gfCNCPoint4[24000] = {X 138.7499, Y 45.9791, Z -6.3333, A 0.000, B 0.000, C 0.000 }
gfCNCPoint4[24001] = {X 138.6396, Y 45.0000, Z -6.3333, A 0.000, B 0.000, C 0.000 }
gfCNCPoint4[24002] = {X 138.6400, Y 44.1483, Z -6.3333, A 0.000, B 0.000, C 0.000 }
gfCNCPoint4[24003] = {X 138.7505, Y 43.2275, Z -6.3333, A 0.000, B 0.000, C 0.000 }
gfCNCPoint4[24004] = {X 139.0514, Y 42.3503, Z -6.3333, A 0.000, B 0.000, C 0.000 }
gfCNCPoint4[24005] = {X 139.5295, Y 41.5556, Z -6.3333, A 0.000, B 0.000, C 0.000 }
gfCNCPoint4[24006] = {X 140.1636, Y 40.8789, Z -6.3333, A 0.000, B 0.000, C 0.000 }
gfCNCPoint4[24007] = {X 140.1636, Y 19.9580, Z -6.3333, A 0.000, B 0.000, C 0.000 }
gfCNCPoint4[24008] = {X 137.4658, Y 19.9576, Z -6.3333, A 0.000, B 0.000, C 0.000 }
gfCNCPoint4[24009] = {X 136.9182, Y 20.6078, Z -6.3333, A 0.000, B 0.000, C 0.000 }
gfCNCPoint4[24010] = {X 136.2556, Y 21.1406, Z -6.3333, A 0.000, B 0.000, C 0.000 }
gfCNCPoint4[24011] = {X 135.5030, Y 21.5361, Z -6.3333, A 0.000, B 0.000, C 0.000 }
gfCNCPoint4[24012] = {X 134.6884, Y 21.7794, Z -6.3333, A 0.000, B 0.000, C 0.000 }
gfCNCPoint4[24013] = {X 133.8422, Y 21.8615, Z -6.3333, A 0.000, B 0.000, C 0.000 }
gfCNCPoint4[24014] = {X 133.2006, Y 21.8615, Z -6.3333, A 0.000, B 0.000, C 0.000 }
gfCNCPoint4[24015] = {X 132.2215, Y 21.7512, Z -6.3333, A 0.000, B 0.000, C 0.000 }
gfCNCPoint4[24016] = {X 131.2916, Y 21.4258, Z -6.3333, A 0.000, B 0.000, C 0.000 }
gfCNCPoint4[24017] = {X 130.4573, Y 20.9016, Z -6.3333, A 0.000, B 0.000, C 0.000 }
gfCNCPoint4[24018] = {X 129.7606, Y 20.2049, Z -6.3333, A 0.000, B 0.000, C 0.000 }
gfCNCPoint4[24019] = {X 129.2364, Y 19.3706, Z -6.3333, A 0.000, B 0.000, C 0.000 }
gfCNCPoint4[24020] = {X 128.9110, Y 18.4406, Z -6.3333, A 0.000, B 0.000, C 0.000 }
gfCNCPoint4[24021] = {X 128.8006, Y 17.4615, Z -6.3333, A 0.000, B 0.000, C 0.000 }
gfCNCPoint4[24022] = {X 128.8006, Y 10.4835, Z -6.3333, A 0.000, B 0.000, C 0.000 }
gfCNCPoint4[24023] = {X 128.8808, Y 9.6474, Z -6.3333, A 0.000, B 0.000, C 0.000 }
gfCNCPoint4[24024] = {X 129.1184, Y 8.8418, Z -6.3333, A 0.000, B 0.000, C 0.000 }
gfCNCPoint4[24025] = {X 129.5047, Y 8.0960, Z -6.3333, A 0.000, B 0.000, C 0.000 }
gfCNCPoint4[24026] = {X 130.0257, Y 7.4372, Z -6.3333, A 0.000, B 0.000, C 0.000 }
gfCNCPoint4[24027] = {X 129.6794, Y 7.1049, Z -6.3333, A 0.000, B 0.000, C 0.000 }
gfCNCPoint4[24028] = {X 102.4337, Y 7.1049, Z -6.3333, A 0.000, B 0.000, C 0.000 }
gfCNCPoint4[24029] = {X 102.4337, Y 11.9049, Z -6.3333, A 0.000, B 0.000, C 0.000 }
gfCNCPoint4[24030] = {X 101.3242, Y 11.9049, Z -6.3333, A 0.000, B 0.000, C 0.000 }
gfCNCPoint4[24031] = {X 101.3283, Y 12.0458, Z -6.3333, A 0.000, B 0.000, C 0.000 }
gfCNCPoint4[24032] = {X 101.3297, Y 12.1868, Z -6.3333, A 0.000, B 0.000, C 0.000 }
gfCNCPoint4[24033] = {X 101.3293, Y 13.0462, Z -6.3333, A 0.000, B 0.000, C 0.000 }
gfCNCPoint4[24034] = {X 101.2275, Y 14.1932, Z -6.3333, A 0.000, B 0.000, C 0.000 }
gfCNCPoint4[24035] = {X 100.9461, Y 15.3098, Z -6.3333, A 0.000, B 0.000, C 0.000 }
gfCNCPoint4[24036] = {X 101.0403, Y 15.5443, Z -6.3333, A 0.000, B 0.000, C 0.000 }
gfCNCPoint4[24037] = {X 101.8677, Y 17.5951, Z -6.3333, A 0.000, B 0.000, C 0.000 }
gfCNCPoint4[24038] = {X 102.7996, Y 15.2734, Z -6.3333, A 0.000, B 0.000, C 0.000 }
gfCNCPoint4[24039] = {X 102.5263, Y 14.1685, Z -6.3333, A 0.000, B 0.000, C 0.000 }
gfCNCPoint4[24040] = {X 102.4285, Y 13.0344, Z -6.3333, A 0.000, B 0.000, C 0.000 }
gfCNCPoint4[24041] = {X 102.4283, Y 12.1868, Z -6.3333, A 0.000, B 0.000, C 0.000 }
gfCNCPoint4[24042] = {X 102.4296, Y 12.0458, Z -6.3333, A 0.000, B 0.000, C 0.000 }
gfCNCPoint4[24043] = {X 102.4337, Y 11.9049, Z -6.3333, A 0.000, B 0.000, C 0.000 }
gfCNCPoint4[24044] = {X 102.4337, Y 9.5049, Z -6.3333, A 0.000, B 0.000, C 0.000 }
gfCNCPoint4[24045] = {X 98.1266, Y 9.5049, Z -6.3333, A 0.000, B 0.000, C 0.000 }
gfCNCPoint4[24046] = {X 98.5429, Y 10.2828, Z -6.3333, A 0.000, B 0.000, C 0.000 }
gfCNCPoint4[24047] = {X 98.8123, Y 11.1229, Z -6.3333, A 0.000, B 0.000, C 0.000 }
gfCNCPoint4[24048] = {X 98.9260, Y 11.9978, Z -6.3333, A 0.000, B 0.000, C 0.000 }
gfCNCPoint4[24049] = {X 98.9288, Y 12.0923, Z -6.3333, A 0.000, B 0.000, C 0.000 }
gfCNCPoint4[24050] = {X 98.9297, Y 12.1868, Z -6.3333, A 0.000, B 0.000, C 0.000 }
gfCNCPoint4[24051] = {X 98.9294, Y 13.0237, Z -6.3333, A 0.000, B 0.000, C 0.000 }
gfCNCPoint4[24052] = {X 98.8590, Y 13.8055, Z -6.3333, A 0.000, B 0.000, C 0.000 }
gfCNCPoint4[24053] = {X 98.6641, Y 14.5659, Z -6.3333, A 0.000, B 0.000, C 0.000 }
gfCNCPoint4[24054] = {X 98.3499, Y 15.2851, Z -6.3333, A 0.000, B 0.000, C 0.000 }
gfCNCPoint4[24055] = {X 98.8140, Y 16.4405, Z -6.3333, A 0.000, B 0.000, C 0.000 }
gfCNCPoint4[24056] = {X 101.8734, Y 24.0244, Z -6.3333, A 0.000, B 0.000, C 0.000 }
gfCNCPoint4[24057] = {X 103.9028, Y 18.9676, Z -6.3333, A 0.000, B 0.000, C 0.000 }
gfCNCPoint4[24058] = {X 105.3927, Y 15.2562, Z -6.3333, A 0.000, B 0.000, C 0.000 }
gfCNCPoint4[24059] = {X 105.0867, Y 14.5450, Z -6.3333, A 0.000, B 0.000, C 0.000 }
gfCNCPoint4[24060] = {X 104.8970, Y 13.7943, Z -6.3333, A 0.000, B 0.000, C 0.000 }
gfCNCPoint4[24061] = {X 104.8285, Y 13.0231, Z -6.3333, A 0.000, B 0.000, C 0.000 }
gfCNCPoint4[24062] = {X 104.8283, Y 12.1868, Z -6.3333, A 0.000, B 0.000, C 0.000 }
gfCNCPoint4[24063] = {X 104.8292, Y 12.0923, Z -6.3333, A 0.000, B 0.000, C 0.000 }
gfCNCPoint4[24064] = {X 104.8319, Y 11.9978, Z -6.3333, A 0.000, B 0.000, C 0.000 }
gfCNCPoint4[24065] = {X 104.9457, Y 11.1229, Z -6.3333, A 0.000, B 0.000, C 0.000 }
gfCNCPoint4[24066] = {X 105.2150, Y 10.2828, Z -6.3333, A 0.000, B 0.000, C 0.000 }
gfCNCPoint4[24067] = {X 105.6313, Y 9.5049, Z -6.3333, A 0.000, B 0.000, C 0.000 }
gfCNCPoint4[24068] = {X 102.4337, Y 9.5049, Z -6.3333, A 0.000, B 0.000, C 0.000 }
gfCNCPoint4[24069] = {X 102.4337, Y 7.1049, Z -6.3333, A 0.000, B 0.000, C 0.000 }
gfCNCPoint4[24070] = {X 64.8349, Y 7.1049, Z -6.3333, A 0.000, B 0.000, C 0.000 }
gfCNCPoint4[24071] = {X 65.5946, Y 8.0241, Z -6.3333, A 0.000, B 0.000, C 0.000 }
gfCNCPoint4[24072] = {X 66.1940, Y 9.0549, Z -6.3333, A 0.000, B 0.000, C 0.000 }
gfCNCPoint4[24073] = {X 66.6171, Y 10.1698, Z -6.3333, A 0.000, B 0.000, C 0.000 }
gfCNCPoint4[24074] = {X 66.8305, Y 11.1683, Z -6.3333, A 0.000, B 0.000, C 0.000 }
gfCNCPoint4[24075] = {X 66.9021, Y 12.1868, Z -6.3333, A 0.000, B 0.000, C 0.000 }
gfCNCPoint4[24076] = {X 66.9018, Y 13.0462, Z -6.3333, A 0.000, B 0.000, C 0.000 }
gfCNCPoint4[24077] = {X 66.7773, Y 14.3204, Z -6.3333, A 0.000, B 0.000, C 0.000 }
gfCNCPoint4[24078] = {X 66.4315, Y 15.5530, Z -6.3333, A 0.000, B 0.000, C 0.000 }
gfCNCPoint4[24079] = {X 74.9126, Y 38.2401, Z -6.3333, A 0.000, B 0.000, C 0.000 }
gfCNCPoint4[24080] = {X 75.8046, Y 38.9749, Z -6.3333, A 0.000, B 0.000, C 0.000 }
gfCNCPoint4[24081] = {X 76.5691, Y 39.8416, Z -6.3333, A 0.000, B 0.000, C 0.000 }
gfCNCPoint4[24082] = {X 77.1868, Y 40.8184, Z -6.3333, A 0.000, B 0.000, C 0.000 }
gfCNCPoint4[24083] = {X 77.6421, Y 41.8806, Z -6.3333, A 0.000, B 0.000, C 0.000 }
gfCNCPoint4[24084] = {X 77.9236, Y 43.0014, Z -6.3333, A 0.000, B 0.000, C 0.000 }
gfCNCPoint4[24085] = {X 78.0243, Y 44.1527, Z -6.3333, A 0.000, B 0.000, C 0.000 }
gfCNCPoint4[24086] = {X 78.0245, Y 45.0000, Z -6.3333, A 0.000, B 0.000, C 0.000 }
gfCNCPoint4[24087] = {X 77.9139, Y 46.2642, Z -6.3333, A 0.000, B 0.000, C 0.000 }
gfCNCPoint4[24088] = {X 77.5854, Y 47.4899, Z -6.3333, A 0.000, B 0.000, C 0.000 }
gfCNCPoint4[24089] = {X 77.0491, Y 48.6400, Z -6.3333, A 0.000, B 0.000, C 0.000 }
gfCNCPoint4[24090] = {X 76.3213, Y 49.6795, Z -6.3333, A 0.000, B 0.000, C 0.000 }
gfCNCPoint4[24091] = {X 75.4240, Y 50.5768, Z -6.3333, A 0.000, B 0.000, C 0.000 }
gfCNCPoint4[24092] = {X 74.3845, Y 51.3047, Z -6.3333, A 0.000, B 0.000, C 0.000 }
gfCNCPoint4[24093] = {X 73.2344, Y 51.8410, Z -6.3333, A 0.000, B 0.000, C 0.000 }
gfCNCPoint4[24094] = {X 72.0086, Y 52.1694, Z -6.3333, A 0.000, B 0.000, C 0.000 }
gfCNCPoint4[24095] = {X 70.7445, Y 52.2800, Z -6.3333, A 0.000, B 0.000, C 0.000 }
gfCNCPoint4[24096] = {X 64.1851, Y 52.2800, Z -6.3333, A 0.000, B 0.000, C 0.000 }
gfCNCPoint4[24097] = {X 62.9397, Y 52.1727, Z -6.3333, A 0.000, B 0.000, C 0.000 }
gfCNCPoint4[24098] = {X 61.7311, Y 51.8539, Z -6.3333, A 0.000, B 0.000, C 0.000 }
gfCNCPoint4[24099] = {X 60.5947, Y 51.3330, Z -6.3333, A 0.000, B 0.000, C 0.000 }
gfCNCPoint4[24100] = {X 59.5643, Y 50.6255, Z -6.3333, A 0.000, B 0.000, C 0.000 }
gfCNCPoint4[24101] = {X 58.6700, Y 49.7521, Z -6.3333, A 0.000, B 0.000, C 0.000 }
gfCNCPoint4[24102] = {X 57.9384, Y 48.7385, Z -6.3333, A 0.000, B 0.000, C 0.000 }
gfCNCPoint4[24103] = {X 57.3706, Y 47.5614, Z -6.3333, A 0.000, B 0.000, C 0.000 }
gfCNCPoint4[24104] = {X 57.0225, Y 46.3017, Z -6.3333, A 0.000, B 0.000, C 0.000 }
gfCNCPoint4[24105] = {X 56.9051, Y 45.0000, Z -6.3333, A 0.000, B 0.000, C 0.000 }
gfCNCPoint4[24106] = {X 56.9052, Y 44.1969, Z -6.3333, A 0.000, B 0.000, C 0.000 }
gfCNCPoint4[24107] = {X 56.9289, Y 43.6212, Z -6.3333, A 0.000, B 0.000, C 0.000 }
gfCNCPoint4[24108] = {X 56.9981, Y 43.0492, Z -6.3333, A 0.000, B 0.000, C 0.000 }
gfCNCPoint4[24109] = {X 54.7600, Y 43.0492, Z -6.3333, A 0.000, B 0.000, C 0.000 }
gfCNCPoint4[24110] = {X 54.8275, Y 43.6012, Z -6.3333, A 0.000, B 0.000, C 0.000 }
gfCNCPoint4[24111] = {X 54.8528, Y 44.1567, Z -6.3333, A 0.000, B 0.000, C 0.000 }
gfCNCPoint4[24112] = {X 54.8529, Y 45.0000, Z -6.3333, A 0.000, B 0.000, C 0.000 }
gfCNCPoint4[24113] = {X 54.7356, Y 46.3017, Z -6.3333, A 0.000, B 0.000, C 0.000 }
gfCNCPoint4[24114] = {X 54.3875, Y 47.5614, Z -6.3333, A 0.000, B 0.000, C 0.000 }
gfCNCPoint4[24115] = {X 53.8197, Y 48.7385, Z -6.3333, A 0.000, B 0.000, C 0.000 }
gfCNCPoint4[24116] = {X 53.0880, Y 49.7521, Z -6.3333, A 0.000, B 0.000, C 0.000 }
gfCNCPoint4[24117] = {X 52.1938, Y 50.6255, Z -6.3333, A 0.000, B 0.000, C 0.000 }
gfCNCPoint4[24118] = {X 51.1633, Y 51.3330, Z -6.3333, A 0.000, B 0.000, C 0.000 }
gfCNCPoint4[24119] = {X 50.0270, Y 51.8539, Z -6.3333, A 0.000, B 0.000, C 0.000 }
gfCNCPoint4[24120] = {X 48.8183, Y 52.1727, Z -6.3333, A 0.000, B 0.000, C 0.000 }
gfCNCPoint4[24121] = {X 47.5729, Y 52.2800, Z -6.3333, A 0.000, B 0.000, C 0.000 }
gfCNCPoint4[24122] = {X 40.6393, Y 52.2800, Z -6.3333, A 0.000, B 0.000, C 0.000 }
gfCNCPoint4[24123] = {X 39.4476, Y 52.1818, Z -6.3333, A 0.000, B 0.000, C 0.000 }
gfCNCPoint4[24124] = {X 38.2881, Y 51.8899, Z -6.3333, A 0.000, B 0.000, C 0.000 }
gfCNCPoint4[24125] = {X 37.1919, Y 51.4120, Z -6.3333, A 0.000, B 0.000, C 0.000 }
gfCNCPoint4[24126] = {X 36.1888, Y 50.7612, Z -6.3333, A 0.000, B 0.000, C 0.000 }
gfCNCPoint4[24127] = {X 35.3058, Y 49.9550, Z -6.3333, A 0.000, B 0.000, C 0.000 }
gfCNCPoint4[24128] = {X 34.8234, Y 50.4196, Z -6.3333, A 0.000, B 0.000, C 0.000 }
gfCNCPoint4[24129] = {X 34.3150, Y 50.8555, Z -6.3333, A 0.000, B 0.000, C 0.000 }
gfCNCPoint4[24130] = {X 33.7788, Y 51.2890, Z -6.3333, A 0.000, B 0.000, C 0.000 }
gfCNCPoint4[24131] = {X 32.5198, Y 52.1756, Z -6.3333, A 0.000, B 0.000, C 0.000 }
gfCNCPoint4[24132] = {X 31.1545, Y 52.8879, Z -6.3333, A 0.000, B 0.000, C 0.000 }
gfCNCPoint4[24133] = {X 29.7070, Y 53.4132, Z -6.3333, A 0.000, B 0.000, C 0.000 }
gfCNCPoint4[24134] = {X 28.2028, Y 53.7423, Z -6.3333, A 0.000, B 0.000, C 0.000 }
gfCNCPoint4[24135] = {X 26.6682, Y 53.8696, Z -6.3333, A 0.000, B 0.000, C 0.000 }
gfCNCPoint4[24136] = {X 24.3194, Y 54.9126, Z -6.3333, A 0.000, B 0.000, C 0.000 }
gfCNCPoint4[24137] = {X 21.9033, Y 55.7884, Z -6.3333, A 0.000, B 0.000, C 0.000 }
gfCNCPoint4[24138] = {X 19.5297, Y 56.4643, Z -6.3333, A 0.000, B 0.000, C 0.000 }
gfCNCPoint4[24139] = {X 17.1086, Y 56.9430, Z -6.3333, A 0.000, B 0.000, C 0.000 }
gfCNCPoint4[24140] = {X 14.6564, Y 57.2213, Z -6.3333, A 0.000, B 0.000, C 0.000 }
gfCNCPoint4[24141] = {X 12.1897, Y 57.2974, Z -6.3333, A 0.000, B 0.000, C 0.000 }
gfCNCPoint4[24142] = {X 9.7250, Y 57.1707, Z -6.3333, A 0.000, B 0.000, C 0.000 }
gfCNCPoint4[24143] = {X 8.4102, Y 57.0194, Z -6.3333, A 0.000, B 0.000, C 0.000 }
gfCNCPoint4[24144] = {X 7.1034, Y 56.8104, Z -6.3333, A 0.000, B 0.000, C 0.000 }
gfCNCPoint4[24145] = {X 7.1034, Y 92.8951, Z -6.3333, A 0.000, B 0.000, C 0.000 }
gfCNCPoint4[24146] = {X 116.2646, Y 92.8951, Z -6.3333, A 0.000, B 0.000, C 0.000 }
gfCNCPoint4[24147] = {X 116.9710, Y 91.6587, Z -6.3333, A 0.000, B 0.000, C 0.000 }
gfCNCPoint4[24148] = {X 117.8511, Y 90.5393, Z -6.3333, A 0.000, B 0.000, C 0.000 }
gfCNCPoint4[24149] = {X 118.8860, Y 89.5612, Z -6.3333, A 0.000, B 0.000, C 0.000 }
gfCNCPoint4[24150] = {X 120.0531, Y 88.7455, Z -6.3333, A 0.000, B 0.000, C 0.000 }
gfCNCPoint4[24151] = {X 121.3272, Y 88.1097, Z -6.3333, A 0.000, B 0.000, C 0.000 }
gfCNCPoint4[24152] = {X 122.6809, Y 87.6678, Z -6.3333, A 0.000, B 0.000, C 0.000 }
gfCNCPoint4[24153] = {X 124.0847, Y 87.4293, Z -6.3333, A 0.000, B 0.000, C 0.000 }
gfCNCPoint4[24154] = {X 124.5363, Y 87.3610, Z -6.3333, A 0.000, B 0.000, C 0.000 }
gfCNCPoint4[24155] = {X 125.0288, Y 86.8573, Z -6.3333, A 0.000, B 0.000, C 0.000 }
gfCNCPoint4[24156] = {X 125.5072, Y 86.3401, Z -6.3333, A 0.000, B 0.000, C 0.000 }
gfCNCPoint4[24157] = {X 149.6585, Y 59.8188, Z -6.3333, A 0.000, B 0.000, C 0.000 }
gfCNCPoint4[24158] = {X 149.6295, Y 59.4063, Z -6.3333, A 0.000, B 0.000, C 0.000 }
gfCNCPoint4[24159] = {X 149.6181, Y 58.9930, Z -6.3333, A 0.000, B 0.000, C 0.000 }
gfCNCPoint4[24160] = {X 149.6180, Y 58.0000, Z -6.3333, A 0.000, B 0.000, C 0.000 }
gfCNCPoint4[24161] = {X 149.6915, Y 56.8093, Z -6.3333, A 0.000, B 0.000, C 0.000 }
gfCNCPoint4[24162] = {X 149.9109, Y 55.6367, Z -6.3333, A 0.000, B 0.000, C 0.000 }
gfCNCPoint4[24163] = {X 150.2729, Y 54.5000, Z -6.3333, A 0.000, B 0.000, C 0.000 }
gfCNCPoint4[24164] = {X 150.7719, Y 53.4164, Z -6.3333, A 0.000, B 0.000, C 0.000 }
gfCNCPoint4[24165] = {X 151.5117, Y 52.2488, Z -6.3333, A 0.000, B 0.000, C 0.000 }
gfCNCPoint4[24166] = {X 152.4103, Y 51.1984, Z -6.3333, A 0.000, B 0.000, C 0.000 }
gfCNCPoint4[24167] = {X 153.4493, Y 50.2867, Z -6.3333, A 0.000, B 0.000, C 0.000 }
gfCNCPoint4[24168] = {X 154.6075, Y 49.5323, Z -6.3333, A 0.000, B 0.000, C 0.000 }
gfCNCPoint4[24169] = {X 155.8614, Y 48.9505, Z -6.3333, A 0.000, B 0.000, C 0.000 }
gfCNCPoint4[24170] = {X 157.1854, Y 48.5533, Z -6.3333, A 0.000, B 0.000, C 0.000 }
gfCNCPoint4[24171] = {X 158.2353, Y 48.3785, Z -6.3333, A 0.000, B 0.000, C 0.000 }
gfCNCPoint4[24172] = {X 159.2980, Y 48.3200, Z -6.3333, A 0.000, B 0.000, C 0.000 }
gfCNCPoint4[24173] = {X 176.3020, Y 48.3200, Z -6.3333, A 0.000, B 0.000, C 0.000 }
gfCNCPoint4[24174] = {X 174.9301, Y 47.4865, Z -6.3333, A 0.000, B 0.000, C 0.000 }
gfCNCPoint4[24175] = {X 173.6422, Y 46.5284, Z -6.3333, A 0.000, B 0.000, C 0.000 }
gfCNCPoint4[24176] = {X 172.5424, Y 45.5341, Z -6.3333, A 0.000, B 0.000, C 0.000 }
gfCNCPoint4[24177] = {X 171.5575, Y 44.4259, Z -6.3333, A 0.000, B 0.000, C 0.000 }
gfCNCPoint4[24178] = {X 170.5960, Y 43.0508, Z -6.3333, A 0.000, B 0.000, C 0.000 }
gfCNCPoint4[24179] = {X 169.8114, Y 41.5676, Z -6.3333, A 0.000, B 0.000, C 0.000 }
gfCNCPoint4[24180] = {X 169.2155, Y 39.9990, Z -6.3333, A 0.000, B 0.000, C 0.000 }
gfCNCPoint4[24181] = {X 168.8176, Y 38.3690, Z -6.3333, A 0.000, B 0.000, C 0.000 }
gfCNCPoint4[24182] = {X 168.7074, Y 37.6766, Z -6.3333, A 0.000, B 0.000, C 0.000 }
gfCNCPoint4[24183] = {X 168.5427, Y 36.0108, Z -6.3333, A 0.000, B 0.000, C 0.000 }
gfCNCPoint4[24184] = {X 168.5600, Y 34.3369, Z -6.3333, A 0.000, B 0.000, C 0.000 }
gfCNCPoint4[24185] = {X 168.7592, Y 32.6747, Z -6.3333, A 0.000, B 0.000, C 0.000 }
gfCNCPoint4[24186] = {X 169.1378, Y 31.0441, Z -6.3333, A 0.000, B 0.000, C 0.000 }
gfCNCPoint4[24187] = {X 169.6914, Y 29.4643, Z -6.3333, A 0.000, B 0.000, C 0.000 }
gfCNCPoint4[24188] = {X 170.2633, Y 28.2675, Z -6.3333, A 0.000, B 0.000, C 0.000 }
gfCNCPoint4[24189] = {X 170.9701, Y 27.1451, Z -6.3333, A 0.000, B 0.000, C 0.000 }
gfCNCPoint4[24190] = {X 171.8024, Y 26.1122, Z -6.3333, A 0.000, B 0.000, C 0.000 }
gfCNCPoint4[24191] = {X 172.7488, Y 25.1829, Z -6.3333, A 0.000, B 0.000, C 0.000 }
gfCNCPoint4[24192] = {X 173.7967, Y 24.3696, Z -6.3333, A 0.000, B 0.000, C 0.000 }
gfCNCPoint4[24193] = {X 173.0267, Y 23.7514, Z -6.3333, A 0.000, B 0.000, C 0.000 }
gfCNCPoint4[24194] = {X 172.3970, Y 22.9909, Z -6.3333, A 0.000, B 0.000, C 0.000 }
gfCNCPoint4[24195] = {X 171.9332, Y 22.1192, Z -6.3333, A 0.000, B 0.000, C 0.000 }
gfCNCPoint4[24196] = {X 169.3220, Y 15.7237, Z -6.3333, A 0.000, B 0.000, C 0.000 }
gfCNCPoint4[24197] = {X 169.1088, Y 15.0753, Z -6.3333, A 0.000, B 0.000, C 0.000 }
gfCNCPoint4[24198] = {X 168.9882, Y 14.4035, Z -6.3333, A 0.000, B 0.000, C 0.000 }
gfCNCPoint4[24199] = {X 168.9599, Y 13.8791, Z -6.3333, A 0.000, B 0.000, C 0.000 }
gfCNCPoint4[24200] = {X 168.9882, Y 13.3548, Z -6.3333, A 0.000, B 0.000, C 0.000 }
gfCNCPoint4[24201] = {X 169.1590, Y 12.4995, Z -6.3333, A 0.000, B 0.000, C 0.000 }
gfCNCPoint4[24202] = {X 169.4794, Y 11.6882, Z -6.3333, A 0.000, B 0.000, C 0.000 }
gfCNCPoint4[24203] = {X 169.9391, Y 10.9470, Z -6.3333, A 0.000, B 0.000, C 0.000 }
gfCNCPoint4[24204] = {X 170.6136, Y 10.2179, Z -6.3333, A 0.000, B 0.000, C 0.000 }
gfCNCPoint4[24205] = {X 171.4217, Y 9.6404, Z -6.3333, A 0.000, B 0.000, C 0.000 }
gfCNCPoint4[24206] = {X 172.0576, Y 9.2779, Z -6.3333, A 0.000, B 0.000, C 0.000 }
gfCNCPoint4[24207] = {X 172.9925, Y 8.8772, Z -6.3333, A 0.000, B 0.000, C 0.000 }
gfCNCPoint4[24208] = {X 173.9903, Y 8.6790, Z -6.3333, A 0.000, B 0.000, C 0.000 }
gfCNCPoint4[24209] = {X 175.0074, Y 8.6919, Z -6.3333, A 0.000, B 0.000, C 0.000 }
gfCNCPoint4[24210] = {X 175.9998, Y 8.9154, Z -6.3333, A 0.000, B 0.000, C 0.000 }
gfCNCPoint4[24211] = {X 176.9280, Y 8.5206, Z -6.3333, A 0.000, B 0.000, C 0.000 }
gfCNCPoint4[24212] = {X 179.1598, Y 7.6998, Z -6.3333, A 0.000, B 0.000, C 0.000 }
gfCNCPoint4[24213] = {X 181.4622, Y 7.1049, Z -6.3333, A 0.000, B 0.000, C 0.000 }
gfCNCPoint4[24214] = {X 168.0206, Y 7.1049, Z -6.3333, A 0.000, B 0.000, C 0.000 }
gfCNCPoint4[24215] = {X 168.0206, Y 4.7049, Z -6.3333, A 0.000, B 0.000, C 0.000 }
gfCNCPoint4[24216] = {X 155.1591, Y 4.7049, Z -6.3333, A 0.000, B 0.000, C 0.000 }
gfCNCPoint4[24217] = {X 155.1591, Y 7.1049, Z -6.3333, A 0.000, B 0.000, C 0.000 }
gfCNCPoint4[24218] = {X 137.3636, Y 7.1049, Z -6.3333, A 0.000, B 0.000, C 0.000 }
gfCNCPoint4[24219] = {X 137.5332, Y 7.2910, Z -6.3333, A 0.000, B 0.000, C 0.000 }
gfCNCPoint4[24220] = {X 137.6930, Y 7.4857, Z -6.3333, A 0.000, B 0.000, C 0.000 }
gfCNCPoint4[24221] = {X 154.8298, Y 7.4857, Z -6.3333, A 0.000, B 0.000, C 0.000 }
gfCNCPoint4[24222] = {X 154.9895, Y 7.2910, Z -6.3333, A 0.000, B 0.000, C 0.000 }
gfCNCPoint4[24223] = {X 155.1591, Y 7.1049, Z -6.3333, A 0.000, B 0.000, C 0.000 }
gfCNCPoint4[24224] = {X 155.1591, Y 4.7049, Z -6.3333, A 0.000, B 0.000, C 0.000 }
gfCNCPoint4[24225] = {X 42.6032, Y 4.7049, Z -6.3333, A 0.000, B 0.000, C 0.000 }
gfCNCPoint4[24226] = {X 42.6032, Y 9.5049, Z -6.3333, A 0.000, B 0.000, C 0.000 }
gfCNCPoint4[24227] = {X 36.0462, Y 9.5049, Z -6.3333, A 0.000, B 0.000, C 0.000 }
gfCNCPoint4[24228] = {X 37.0562, Y 11.3879, Z -6.3333, A 0.000, B 0.000, C 0.000 }
gfCNCPoint4[24229] = {X 37.8845, Y 13.3577, Z -6.3333, A 0.000, B 0.000, C 0.000 }
gfCNCPoint4[24230] = {X 38.5471, Y 15.5383, Z -6.3333, A 0.000, B 0.000, C 0.000 }
gfCNCPoint4[24231] = {X 39.0057, Y 17.7709, Z -6.3333, A 0.000, B 0.000, C 0.000 }
gfCNCPoint4[24232] = {X 39.2564, Y 20.0362, Z -6.3333, A 0.000, B 0.000, C 0.000 }
gfCNCPoint4[24233] = {X 39.2971, Y 22.3149, Z -6.3333, A 0.000, B 0.000, C 0.000 }
gfCNCPoint4[24234] = {X 39.1274, Y 24.5877, Z -6.3333, A 0.000, B 0.000, C 0.000 }
gfCNCPoint4[24235] = {X 42.5394, Y 15.4279, Z -6.3333, A 0.000, B 0.000, C 0.000 }
gfCNCPoint4[24236] = {X 42.3075, Y 14.2452, Z -6.3333, A 0.000, B 0.000, C 0.000 }
gfCNCPoint4[24237] = {X 42.2244, Y 13.0428, Z -6.3333, A 0.000, B 0.000, C 0.000 }
gfCNCPoint4[24238] = {X 42.2242, Y 12.1868, Z -6.3333, A 0.000, B 0.000, C 0.000 }
gfCNCPoint4[24239] = {X 42.3194, Y 10.8325, Z -6.3333, A 0.000, B 0.000, C 0.000 }
gfCNCPoint4[24240] = {X 42.6032, Y 9.5049, Z -6.3333, A 0.000, B 0.000, C 0.000 }
gfCNCPoint4[24241] = {X 42.6032, Y 7.1049, Z -6.3333, A 0.000, B 0.000, C 0.000 }
gfCNCPoint4[24242] = {X 31.2118, Y 7.1049, Z -6.3333, A 0.000, B 0.000, C 0.000 }
gfCNCPoint4[24243] = {X 32.2273, Y 8.2449, Z -6.3333, A 0.000, B 0.000, C 0.000 }
gfCNCPoint4[24244] = {X 33.1541, Y 9.4582, Z -6.3333, A 0.000, B 0.000, C 0.000 }
gfCNCPoint4[24245] = {X 33.9870, Y 10.7376, Z -6.3333, A 0.000, B 0.000, C 0.000 }
gfCNCPoint4[24246] = {X 34.8876, Y 12.4162, Z -6.3333, A 0.000, B 0.000, C 0.000 }
gfCNCPoint4[24247] = {X 35.6267, Y 14.1718, Z -6.3333, A 0.000, B 0.000, C 0.000 }
gfCNCPoint4[24248] = {X 36.2233, Y 16.1384, Z -6.3333, A 0.000, B 0.000, C 0.000 }
gfCNCPoint4[24249] = {X 36.6361, Y 18.1517, Z -6.3333, A 0.000, B 0.000, C 0.000 }
gfCNCPoint4[24250] = {X 36.8616, Y 20.1944, Z -6.3333, A 0.000, B 0.000, C 0.000 }
gfCNCPoint4[24251] = {X 36.8980, Y 22.2492, Z -6.3333, A 0.000, B 0.000, C 0.000 }
gfCNCPoint4[24252] = {X 36.7448, Y 24.2987, Z -6.3333, A 0.000, B 0.000, C 0.000 }
gfCNCPoint4[24253] = {X 36.5515, Y 25.5796, Z -6.3333, A 0.000, B 0.000, C 0.000 }
gfCNCPoint4[24254] = {X 36.2840, Y 26.8471, Z -6.3333, A 0.000, B 0.000, C 0.000 }
gfCNCPoint4[24255] = {X 35.8750, Y 28.3066, Z -6.3333, A 0.000, B 0.000, C 0.000 }
gfCNCPoint4[24256] = {X 35.3508, Y 29.7287, Z -6.3333, A 0.000, B 0.000, C 0.000 }
gfCNCPoint4[24257] = {X 34.7147, Y 31.1045, Z -6.3333, A 0.000, B 0.000, C 0.000 }
gfCNCPoint4[24258] = {X 37.2840, Y 36.4121, Z -6.3333, A 0.000, B 0.000, C 0.000 }
gfCNCPoint4[24259] = {X 41.3764, Y 25.4255, Z -6.3333, A 0.000, B 0.000, C 0.000 }
gfCNCPoint4[24260] = {X 45.0743, Y 15.4981, Z -6.3333, A 0.000, B 0.000, C 0.000 }
gfCNCPoint4[24261] = {X 44.7425, Y 14.2852, Z -6.3333, A 0.000, B 0.000, C 0.000 }
gfCNCPoint4[24262] = {X 44.6244, Y 13.0334, Z -6.3333, A 0.000, B 0.000, C 0.000 }
gfCNCPoint4[24263] = {X 44.6242, Y 12.1868, Z -6.3333, A 0.000, B 0.000, C 0.000 }
gfCNCPoint4[24264] = {X 44.6958, Y 11.1683, Z -6.3333, A 0.000, B 0.000, C 0.000 }
gfCNCPoint4[24265] = {X 44.9092, Y 10.1698, Z -6.3333, A 0.000, B 0.000, C 0.000 }
gfCNCPoint4[24266] = {X 45.3323, Y 9.0549, Z -6.3333, A 0.000, B 0.000, C 0.000 }
gfCNCPoint4[24267] = {X 45.9318, Y 8.0241, Z -6.3333, A 0.000, B 0.000, C 0.000 }
gfCNCPoint4[24268] = {X 46.6915, Y 7.1049, Z -6.3333, A 0.000, B 0.000, C 0.000 }
gfCNCPoint4[24269] = {X 42.6032, Y 7.1049, Z -6.3333, A 0.000, B 0.000, C 0.000 }
gfCNCPoint4[24270] = {X 42.6032, Y 4.7049, Z -6.3333, A 0.000, B 0.000, C 0.000 }
gfCNCPoint4[24271] = {X 23.8365, Y 4.7049, Z -6.3333, A 0.000, B 0.000, C 0.000 }
gfCNCPoint4[24272] = {X 25.7643, Y 5.7847, Z -6.3333, A 0.000, B 0.000, C 0.000 }
gfCNCPoint4[24273] = {X 27.5759, Y 7.0498, Z -6.3333, A 0.000, B 0.000, C 0.000 }
gfCNCPoint4[24274] = {X 28.5593, Y 7.8745, Z -6.3333, A 0.000, B 0.000, C 0.000 }
gfCNCPoint4[24275] = {X 29.4810, Y 8.7675, Z -6.3333, A 0.000, B 0.000, C 0.000 }
gfCNCPoint4[24276] = {X 30.6893, Y 10.1628, Z -6.3333, A 0.000, B 0.000, C 0.000 }
gfCNCPoint4[24277] = {X 31.7473, Y 11.6753, Z -6.3333, A 0.000, B 0.000, C 0.000 }
gfCNCPoint4[24278] = {X 32.6437, Y 13.2887, Z -6.3333, A 0.000, B 0.000, C 0.000 }
gfCNCPoint4[24279] = {X 33.3690, Y 14.9860, Z -6.3333, A 0.000, B 0.000, C 0.000 }
gfCNCPoint4[24280] = {X 33.9192, Y 16.8170, Z -6.3333, A 0.000, B 0.000, C 0.000 }
gfCNCPoint4[24281] = {X 34.2909, Y 18.6923, Z -6.3333, A 0.000, B 0.000, C 0.000 }
gfCNCPoint4[24282] = {X 34.4808, Y 20.5947, Z -6.3333, A 0.000, B 0.000, C 0.000 }
gfCNCPoint4[24283] = {X 34.4870, Y 22.5066, Z -6.3333, A 0.000, B 0.000, C 0.000 }
gfCNCPoint4[24284] = {X 34.3096, Y 24.4102, Z -6.3333, A 0.000, B 0.000, C 0.000 }
gfCNCPoint4[24285] = {X 33.9501, Y 26.2879, Z -6.3333, A 0.000, B 0.000, C 0.000 }
gfCNCPoint4[24286] = {X 33.4662, Y 27.9397, Z -6.3333, A 0.000, B 0.000, C 0.000 }
gfCNCPoint4[24287] = {X 32.8137, Y 29.5323, Z -6.3333, A 0.000, B 0.000, C 0.000 }
gfCNCPoint4[24288] = {X 31.9994, Y 31.0487, Z -6.3333, A 0.000, B 0.000, C 0.000 }
gfCNCPoint4[24289] = {X 32.1288, Y 31.2844, Z -6.3333, A 0.000, B 0.000, C 0.000 }
gfCNCPoint4[24290] = {X 32.2513, Y 31.5237, Z -6.3333, A 0.000, B 0.000, C 0.000 }
gfCNCPoint4[24291] = {X 35.3025, Y 37.8269, Z -6.3333, A 0.000, B 0.000, C 0.000 }
gfCNCPoint4[24292] = {X 35.7263, Y 38.8573, Z -6.3333, A 0.000, B 0.000, C 0.000 }
gfCNCPoint4[24293] = {X 36.0224, Y 39.9313, Z -6.3333, A 0.000, B 0.000, C 0.000 }
gfCNCPoint4[24294] = {X 36.1865, Y 41.0332, Z -6.3333, A 0.000, B 0.000, C 0.000 }
gfCNCPoint4[24295] = {X 36.2163, Y 42.1469, Z -6.3333, A 0.000, B 0.000, C 0.000 }
gfCNCPoint4[24296] = {X 36.6303, Y 41.4264, Z -6.3333, A 0.000, B 0.000, C 0.000 }
gfCNCPoint4[24297] = {X 37.1605, Y 40.7865, Z -6.3333, A 0.000, B 0.000, C 0.000 }
gfCNCPoint4[24298] = {X 37.7916, Y 40.2458, Z -6.3333, A 0.000, B 0.000, C 0.000 }
gfCNCPoint4[24299] = {X 38.5053, Y 39.8201, Z -6.3333, A 0.000, B 0.000, C 0.000 }
gfCNCPoint4[24300] = {X 39.0443, Y 38.5343, Z -6.3333, A 0.000, B 0.000, C 0.000 }
gfCNCPoint4[24301] = {X 39.5399, Y 37.2311, Z -6.3333, A 0.000, B 0.000, C 0.000 }
gfCNCPoint4[24302] = {X 47.6702, Y 15.4045, Z -6.3333, A 0.000, B 0.000, C 0.000 }
gfCNCPoint4[24303] = {X 47.3200, Y 14.6512, Z -6.3333, A 0.000, B 0.000, C 0.000 }
gfCNCPoint4[24304] = {X 47.1026, Y 13.8493, Z -6.3333, A 0.000, B 0.000, C 0.000 }
gfCNCPoint4[24305] = {X 47.0244, Y 13.0222, Z -6.3333, A 0.000, B 0.000, C 0.000 }
gfCNCPoint4[24306] = {X 47.0242, Y 12.1868, Z -6.3333, A 0.000, B 0.000, C 0.000 }
gfCNCPoint4[24307] = {X 47.1150, Y 11.2500, Z -6.3333, A 0.000, B 0.000, C 0.000 }
gfCNCPoint4[24308] = {X 47.3839, Y 10.3480, Z -6.3333, A 0.000, B 0.000, C 0.000 }
gfCNCPoint4[24309] = {X 47.8210, Y 9.5144, Z -6.3333, A 0.000, B 0.000, C 0.000 }
gfCNCPoint4[24310] = {X 48.4100, Y 8.7803, Z -6.3333, A 0.000, B 0.000, C 0.000 }
gfCNCPoint4[24311] = {X 49.1545, Y 8.1553, Z -6.3333, A 0.000, B 0.000, C 0.000 }
gfCNCPoint4[24312] = {X 50.0081, Y 7.6902, Z -6.3333, A 0.000, B 0.000, C 0.000 }
gfCNCPoint4[24313] = {X 50.9370, Y 7.4036, Z -6.3333, A 0.000, B 0.000, C 0.000 }
gfCNCPoint4[24314] = {X 51.9042, Y 7.3068, Z -6.3333, A 0.000, B 0.000, C 0.000 }
gfCNCPoint4[24315] = {X 59.6221, Y 7.3068, Z -6.3333, A 0.000, B 0.000, C 0.000 }
gfCNCPoint4[24316] = {X 60.5894, Y 7.4036, Z -6.3333, A 0.000, B 0.000, C 0.000 }
gfCNCPoint4[24317] = {X 61.5182, Y 7.6902, Z -6.3333, A 0.000, B 0.000, C 0.000 }
gfCNCPoint4[24318] = {X 62.3719, Y 8.1553, Z -6.3333, A 0.000, B 0.000, C 0.000 }
gfCNCPoint4[24319] = {X 63.1164, Y 8.7803, Z -6.3333, A 0.000, B 0.000, C 0.000 }
gfCNCPoint4[24320] = {X 63.7053, Y 9.5144, Z -6.3333, A 0.000, B 0.000, C 0.000 }
gfCNCPoint4[24321] = {X 64.1424, Y 10.3480, Z -6.3333, A 0.000, B 0.000, C 0.000 }
gfCNCPoint4[24322] = {X 64.4114, Y 11.2500, Z -6.3333, A 0.000, B 0.000, C 0.000 }
gfCNCPoint4[24323] = {X 64.5021, Y 12.1868, Z -6.3333, A 0.000, B 0.000, C 0.000 }
gfCNCPoint4[24324] = {X 64.5019, Y 13.0237, Z -6.3333, A 0.000, B 0.000, C 0.000 }
gfCNCPoint4[24325] = {X 64.4204, Y 13.8671, Z -6.3333, A 0.000, B 0.000, C 0.000 }
gfCNCPoint4[24326] = {X 64.1943, Y 14.6837, Z -6.3333, A 0.000, B 0.000, C 0.000 }
gfCNCPoint4[24327] = {X 63.8304, Y 15.4489, Z -6.3333, A 0.000, B 0.000, C 0.000 }
gfCNCPoint4[24328] = {X 72.9553, Y 39.8583, Z -6.3333, A 0.000, B 0.000, C 0.000 }
gfCNCPoint4[24329] = {X 73.8450, Y 40.4403, Z -6.3333, A 0.000, B 0.000, C 0.000 }
gfCNCPoint4[24330] = {X 74.5875, Y 41.2012, Z -6.3333, A 0.000, B 0.000, C 0.000 }
gfCNCPoint4[24331] = {X 75.1476, Y 42.1048, Z -6.3333, A 0.000, B 0.000, C 0.000 }
gfCNCPoint4[24332] = {X 75.4988, Y 43.1083, Z -6.3333, A 0.000, B 0.000, C 0.000 }
gfCNCPoint4[24333] = {X 75.6243, Y 44.1640, Z -6.3333, A 0.000, B 0.000, C 0.000 }
gfCNCPoint4[24334] = {X 75.6245, Y 45.0000, Z -6.3333, A 0.000, B 0.000, C 0.000 }
gfCNCPoint4[24335] = {X 75.5307, Y 45.9520, Z -6.3333, A 0.000, B 0.000, C 0.000 }
gfCNCPoint4[24336] = {X 75.2530, Y 46.8675, Z -6.3333, A 0.000, B 0.000, C 0.000 }
gfCNCPoint4[24337] = {X 74.8020, Y 47.7112, Z -6.3333, A 0.000, B 0.000, C 0.000 }
gfCNCPoint4[24338] = {X 74.1951, Y 48.4507, Z -6.3333, A 0.000, B 0.000, C 0.000 }
gfCNCPoint4[24339] = {X 73.4556, Y 49.0576, Z -6.3333, A 0.000, B 0.000, C 0.000 }
gfCNCPoint4[24340] = {X 72.6120, Y 49.5085, Z -6.3333, A 0.000, B 0.000, C 0.000 }
gfCNCPoint4[24341] = {X 71.6965, Y 49.7862, Z -6.3333, A 0.000, B 0.000, C 0.000 }
gfCNCPoint4[24342] = {X 70.7445, Y 49.8800, Z -6.3333, A 0.000, B 0.000, C 0.000 }
gfCNCPoint4[24343] = {X 64.1851, Y 49.8800, Z -6.3333, A 0.000, B 0.000, C 0.000 }
gfCNCPoint4[24344] = {X 63.2331, Y 49.7862, Z -6.3333, A 0.000, B 0.000, C 0.000 }
gfCNCPoint4[24345] = {X 62.3176, Y 49.5085, Z -6.3333, A 0.000, B 0.000, C 0.000 }
gfCNCPoint4[24346] = {X 61.4740, Y 49.0576, Z -6.3333, A 0.000, B 0.000, C 0.000 }
gfCNCPoint4[24347] = {X 60.7345, Y 48.4507, Z -6.3333, A 0.000, B 0.000, C 0.000 }
gfCNCPoint4[24348] = {X 60.1276, Y 47.7112, Z -6.3333, A 0.000, B 0.000, C 0.000 }
gfCNCPoint4[24349] = {X 59.6766, Y 46.8675, Z -6.3333, A 0.000, B 0.000, C 0.000 }
gfCNCPoint4[24350] = {X 59.3989, Y 45.9520, Z -6.3333, A 0.000, B 0.000, C 0.000 }
gfCNCPoint4[24351] = {X 59.3051, Y 45.0000, Z -6.3333, A 0.000, B 0.000, C 0.000 }
gfCNCPoint4[24352] = {X 59.3052, Y 44.2028, Z -6.3333, A 0.000, B 0.000, C 0.000 }
gfCNCPoint4[24353] = {X 59.3847, Y 43.3313, Z -6.3333, A 0.000, B 0.000, C 0.000 }
gfCNCPoint4[24354] = {X 59.6186, Y 42.4880, Z -6.3333, A 0.000, B 0.000, C 0.000 }
gfCNCPoint4[24355] = {X 59.9994, Y 41.7000, Z -6.3333, A 0.000, B 0.000, C 0.000 }
gfCNCPoint4[24356] = {X 59.6152, Y 40.6492, Z -6.3333, A 0.000, B 0.000, C 0.000 }
gfCNCPoint4[24357] = {X 52.4670, Y 40.6492, Z -6.3333, A 0.000, B 0.000, C 0.000 }
gfCNCPoint4[24358] = {X 51.9473, Y 42.0456, Z -6.3333, A 0.000, B 0.000, C 0.000 }
gfCNCPoint4[24359] = {X 52.2218, Y 42.7247, Z -6.3333, A 0.000, B 0.000, C 0.000 }
gfCNCPoint4[24360] = {X 52.3916, Y 43.4373, Z -6.3333, A 0.000, B 0.000, C 0.000 }
gfCNCPoint4[24361] = {X 52.4528, Y 44.1672, Z -6.3333, A 0.000, B 0.000, C 0.000 }
gfCNCPoint4[24362] = {X 52.4529, Y 45.0000, Z -6.3333, A 0.000, B 0.000, C 0.000 }
gfCNCPoint4[24363] = {X 52.3592, Y 45.9520, Z -6.3333, A 0.000, B 0.000, C 0.000 }
gfCNCPoint4[24364] = {X 52.0815, Y 46.8675, Z -6.3333, A 0.000, B 0.000, C 0.000 }
gfCNCPoint4[24365] = {X 51.6305, Y 47.7112, Z -6.3333, A 0.000, B 0.000, C 0.000 }
gfCNCPoint4[24366] = {X 51.0236, Y 48.4507, Z -6.3333, A 0.000, B 0.000, C 0.000 }
gfCNCPoint4[24367] = {X 50.2841, Y 49.0576, Z -6.3333, A 0.000, B 0.000, C 0.000 }
gfCNCPoint4[24368] = {X 49.4404, Y 49.5085, Z -6.3333, A 0.000, B 0.000, C 0.000 }
gfCNCPoint4[24369] = {X 48.5250, Y 49.7862, Z -6.3333, A 0.000, B 0.000, C 0.000 }
gfCNCPoint4[24370] = {X 47.5729, Y 49.8800, Z -6.3333, A 0.000, B 0.000, C 0.000 }
gfCNCPoint4[24371] = {X 40.6393, Y 49.8800, Z -6.3333, A 0.000, B 0.000, C 0.000 }
gfCNCPoint4[24372] = {X 39.6433, Y 49.7773, Z -6.3333, A 0.000, B 0.000, C 0.000 }
gfCNCPoint4[24373] = {X 38.6892, Y 49.4734, Z -6.3333, A 0.000, B 0.000, C 0.000 }
gfCNCPoint4[24374] = {X 37.8173, Y 48.9813, Z -6.3333, A 0.000, B 0.000, C 0.000 }
gfCNCPoint4[24375] = {X 37.0641, Y 48.3215, Z -6.3333, A 0.000, B 0.000, C 0.000 }
gfCNCPoint4[24376] = {X 36.5085, Y 47.5983, Z -6.3333, A 0.000, B 0.000, C 0.000 }
gfCNCPoint4[24377] = {X 36.0972, Y 46.7843, Z -6.3333, A 0.000, B 0.000, C 0.000 }
gfCNCPoint4[24378] = {X 35.8445, Y 45.9080, Z -6.3333, A 0.000, B 0.000, C 0.000 }
gfCNCPoint4[24379] = {X 35.7593, Y 45.0000, Z -6.3333, A 0.000, B 0.000, C 0.000 }
gfCNCPoint4[24380] = {X 35.7593, Y 44.7148, Z -6.3333, A 0.000, B 0.000, C 0.000 }
gfCNCPoint4[24381] = {X 36.2393, Y 44.7148, Z -6.3333, A 0.000, B 0.000, C 0.000 }
gfCNCPoint4[24382] = {X 36.2397, Y 44.1483, Z -6.3333, A 0.000, B 0.000, C 0.000 }
gfCNCPoint4[24383] = {X 36.3680, Y 43.1524, Z -6.3333, A 0.000, B 0.000, C 0.000 }
gfCNCPoint4[24384] = {X 36.7187, Y 42.2115, Z -6.3333, A 0.000, B 0.000, C 0.000 }
gfCNCPoint4[24385] = {X 37.2737, Y 41.3746, Z -6.3333, A 0.000, B 0.000, C 0.000 }
gfCNCPoint4[24386] = {X 38.0039, Y 40.6854, Z -6.3333, A 0.000, B 0.000, C 0.000 }
gfCNCPoint4[24387] = {X 38.8713, Y 40.1796, Z -6.3333, A 0.000, B 0.000, C 0.000 }
gfCNCPoint4[24388] = {X 39.4552, Y 38.7991, Z -6.3333, A 0.000, B 0.000, C 0.000 }
gfCNCPoint4[24389] = {X 39.9897, Y 37.3987, Z -6.3333, A 0.000, B 0.000, C 0.000 }
gfCNCPoint4[24390] = {X 48.2011, Y 15.3544, Z -6.3333, A 0.000, B 0.000, C 0.000 }
gfCNCPoint4[24391] = {X 47.8187, Y 14.6115, Z -6.3333, A 0.000, B 0.000, C 0.000 }
gfCNCPoint4[24392] = {X 47.5835, Y 13.8097, Z -6.3333, A 0.000, B 0.000, C 0.000 }
gfCNCPoint4[24393] = {X 47.5042, Y 12.9780, Z -6.3333, A 0.000, B 0.000, C 0.000 }
gfCNCPoint4[24394] = {X 47.5042, Y 12.1868, Z -6.3333, A 0.000, B 0.000, C 0.000 }
gfCNCPoint4[24395] = {X 47.6145, Y 11.2077, Z -6.3333, A 0.000, B 0.000, C 0.000 }
gfCNCPoint4[24396] = {X 47.9400, Y 10.2777, Z -6.3333, A 0.000, B 0.000, C 0.000 }
gfCNCPoint4[24397] = {X 48.4642, Y 9.4435, Z -6.3333, A 0.000, B 0.000, C 0.000 }
gfCNCPoint4[24398] = {X 49.1609, Y 8.7468, Z -6.3333, A 0.000, B 0.000, C 0.000 }
gfCNCPoint4[24399] = {X 49.9951, Y 8.2226, Z -6.3333, A 0.000, B 0.000, C 0.000 }
gfCNCPoint4[24400] = {X 50.9251, Y 7.8971, Z -6.3333, A 0.000, B 0.000, C 0.000 }
gfCNCPoint4[24401] = {X 51.9042, Y 7.7868, Z -6.3333, A 0.000, B 0.000, C 0.000 }
gfCNCPoint4[24402] = {X 59.6221, Y 7.7868, Z -6.3333, A 0.000, B 0.000, C 0.000 }
gfCNCPoint4[24403] = {X 60.6012, Y 7.8971, Z -6.3333, A 0.000, B 0.000, C 0.000 }
gfCNCPoint4[24404] = {X 61.5312, Y 8.2226, Z -6.3333, A 0.000, B 0.000, C 0.000 }
gfCNCPoint4[24405] = {X 62.3655, Y 8.7468, Z -6.3333, A 0.000, B 0.000, C 0.000 }
gfCNCPoint4[24406] = {X 63.0622, Y 9.4435, Z -6.3333, A 0.000, B 0.000, C 0.000 }
gfCNCPoint4[24407] = {X 63.5864, Y 10.2777, Z -6.3333, A 0.000, B 0.000, C 0.000 }
gfCNCPoint4[24408] = {X 63.9118, Y 11.2077, Z -6.3333, A 0.000, B 0.000, C 0.000 }
gfCNCPoint4[24409] = {X 64.0221, Y 12.1868, Z -6.3333, A 0.000, B 0.000, C 0.000 }
gfCNCPoint4[24410] = {X 64.0219, Y 13.0233, Z -6.3333, A 0.000, B 0.000, C 0.000 }
gfCNCPoint4[24411] = {X 63.9336, Y 13.8561, Z -6.3333, A 0.000, B 0.000, C 0.000 }
gfCNCPoint4[24412] = {X 63.6892, Y 14.6570, Z -6.3333, A 0.000, B 0.000, C 0.000 }
gfCNCPoint4[24413] = {X 63.2974, Y 15.3971, Z -6.3333, A 0.000, B 0.000, C 0.000 }
gfCNCPoint4[24414] = {X 63.5014, Y 15.9354, Z -6.3333, A 0.000, B 0.000, C 0.000 }
gfCNCPoint4[24415] = {X 66.3154, Y 23.4033, Z -6.3333, A 0.000, B 0.000, C 0.000 }
gfCNCPoint4[24416] = {X 72.2850, Y 39.4717, Z -6.3333, A 0.000, B 0.000, C 0.000 }
gfCNCPoint4[24417] = {X 72.5782, Y 40.2091, Z -6.3333, A 0.000, B 0.000, C 0.000 }
gfCNCPoint4[24418] = {X 73.4354, Y 40.7276, Z -6.3333, A 0.000, B 0.000, C 0.000 }
gfCNCPoint4[24419] = {X 74.1532, Y 41.4266, Z -6.3333, A 0.000, B 0.000, C 0.000 }
gfCNCPoint4[24420] = {X 74.6942, Y 42.2698, Z -6.3333, A 0.000, B 0.000, C 0.000 }
gfCNCPoint4[24421] = {X 75.0304, Y 43.2135, Z -6.3333, A 0.000, B 0.000, C 0.000 }
gfCNCPoint4[24422] = {X 75.1445, Y 44.2089, Z -6.3333, A 0.000, B 0.000, C 0.000 }
gfCNCPoint4[24423] = {X 75.1445, Y 45.0000, Z -6.3333, A 0.000, B 0.000, C 0.000 }
gfCNCPoint4[24424] = {X 75.0341, Y 45.9791, Z -6.3333, A 0.000, B 0.000, C 0.000 }
gfCNCPoint4[24425] = {X 74.7087, Y 46.9091, Z -6.3333, A 0.000, B 0.000, C 0.000 }
gfCNCPoint4[24426] = {X 74.1845, Y 47.7434, Z -6.3333, A 0.000, B 0.000, C 0.000 }
gfCNCPoint4[24427] = {X 73.4878, Y 48.4401, Z -6.3333, A 0.000, B 0.000, C 0.000 }
gfCNCPoint4[24428] = {X 72.6535, Y 48.9643, Z -6.3333, A 0.000, B 0.000, C 0.000 }
gfCNCPoint4[24429] = {X 71.7236, Y 49.2897, Z -6.3333, A 0.000, B 0.000, C 0.000 }
gfCNCPoint4[24430] = {X 70.7445, Y 49.4000, Z -6.3333, A 0.000, B 0.000, C 0.000 }
gfCNCPoint4[24431] = {X 64.1851, Y 49.4000, Z -6.3333, A 0.000, B 0.000, C 0.000 }
gfCNCPoint4[24432] = {X 63.2060, Y 49.2897, Z -6.3333, A 0.000, B 0.000, C 0.000 }
gfCNCPoint4[24433] = {X 62.2760, Y 48.9643, Z -6.3333, A 0.000, B 0.000, C 0.000 }
gfCNCPoint4[24434] = {X 61.4418, Y 48.4401, Z -6.3333, A 0.000, B 0.000, C 0.000 }
gfCNCPoint4[24435] = {X 60.7451, Y 47.7434, Z -6.3333, A 0.000, B 0.000, C 0.000 }
gfCNCPoint4[24436] = {X 60.2209, Y 46.9091, Z -6.3333, A 0.000, B 0.000, C 0.000 }
gfCNCPoint4[24437] = {X 59.8955, Y 45.9791, Z -6.3333, A 0.000, B 0.000, C 0.000 }
gfCNCPoint4[24438] = {X 59.7851, Y 45.0000, Z -6.3333, A 0.000, B 0.000, C 0.000 }
gfCNCPoint4[24439] = {X 59.7856, Y 44.1483, Z -6.3333, A 0.000, B 0.000, C 0.000 }
gfCNCPoint4[24440] = {X 59.8783, Y 43.3081, Z -6.3333, A 0.000, B 0.000, C 0.000 }
gfCNCPoint4[24441] = {X 60.1300, Y 42.5011, Z -6.3333, A 0.000, B 0.000, C 0.000 }
gfCNCPoint4[24442] = {X 60.5314, Y 41.7572, Z -6.3333, A 0.000, B 0.000, C 0.000 }
gfCNCPoint4[24443] = {X 59.9507, Y 40.1692, Z -6.3333, A 0.000, B 0.000, C 0.000 }
gfCNCPoint4[24444] = {X 52.1335, Y 40.1692, Z -6.3333, A 0.000, B 0.000, C 0.000 }
gfCNCPoint4[24445] = {X 51.4229, Y 42.0785, Z -6.3333, A 0.000, B 0.000, C 0.000 }
gfCNCPoint4[24446] = {X 51.7256, Y 42.7542, Z -6.3333, A 0.000, B 0.000, C 0.000 }
gfCNCPoint4[24447] = {X 51.9107, Y 43.4711, Z -6.3333, A 0.000, B 0.000, C 0.000 }
gfCNCPoint4[24448] = {X 51.9729, Y 44.2089, Z -6.3333, A 0.000, B 0.000, C 0.000 }
gfCNCPoint4[24449] = {X 51.9729, Y 45.0000, Z -6.3333, A 0.000, B 0.000, C 0.000 }
gfCNCPoint4[24450] = {X 51.8626, Y 45.9791, Z -6.3333, A 0.000, B 0.000, C 0.000 }
gfCNCPoint4[24451] = {X 51.5372, Y 46.9091, Z -6.3333, A 0.000, B 0.000, C 0.000 }
gfCNCPoint4[24452] = {X 51.0130, Y 47.7434, Z -6.3333, A 0.000, B 0.000, C 0.000 }
gfCNCPoint4[24453] = {X 50.3163, Y 48.4401, Z -6.3333, A 0.000, B 0.000, C 0.000 }
gfCNCPoint4[24454] = {X 49.4820, Y 48.9643, Z -6.3333, A 0.000, B 0.000, C 0.000 }
gfCNCPoint4[24455] = {X 48.5520, Y 49.2897, Z -6.3333, A 0.000, B 0.000, C 0.000 }
gfCNCPoint4[24456] = {X 47.5729, Y 49.4000, Z -6.3333, A 0.000, B 0.000, C 0.000 }
gfCNCPoint4[24457] = {X 40.6393, Y 49.4000, Z -6.3333, A 0.000, B 0.000, C 0.000 }
gfCNCPoint4[24458] = {X 39.6602, Y 49.2897, Z -6.3333, A 0.000, B 0.000, C 0.000 }
gfCNCPoint4[24459] = {X 38.7302, Y 48.9643, Z -6.3333, A 0.000, B 0.000, C 0.000 }
gfCNCPoint4[24460] = {X 37.8959, Y 48.4401, Z -6.3333, A 0.000, B 0.000, C 0.000 }
gfCNCPoint4[24461] = {X 37.1992, Y 47.7434, Z -6.3333, A 0.000, B 0.000, C 0.000 }
gfCNCPoint4[24462] = {X 36.6750, Y 46.9091, Z -6.3333, A 0.000, B 0.000, C 0.000 }
gfCNCPoint4[24463] = {X 36.3496, Y 45.9791, Z -6.3333, A 0.000, B 0.000, C 0.000 }
gfCNCPoint4[24464] = {X 36.2393, Y 45.0000, Z -6.3333, A 0.000, B 0.000, C 0.000 }
gfCNCPoint4[24465] = {X 36.2393, Y 44.7148, Z -6.3333, A 0.000, B 0.000, C 0.000 }
gfCNCPoint4[24466] = {X 35.7593, Y 44.7148, Z -6.3333, A 0.000, B 0.000, C 0.000 }
gfCNCPoint4[24467] = {X 35.2211, Y 46.0074, Z -6.3333, A 0.000, B 0.000, C 0.000 }
gfCNCPoint4[24468] = {X 34.4930, Y 47.2034, Z -6.3333, A 0.000, B 0.000, C 0.000 }
gfCNCPoint4[24469] = {X 33.5918, Y 48.2750, Z -6.3333, A 0.000, B 0.000, C 0.000 }
gfCNCPoint4[24470] = {X 33.2092, Y 48.6435, Z -6.3333, A 0.000, B 0.000, C 0.000 }
gfCNCPoint4[24471] = {X 32.8060, Y 48.9892, Z -6.3333, A 0.000, B 0.000, C 0.000 }
gfCNCPoint4[24472] = {X 32.2699, Y 49.4227, Z -6.3333, A 0.000, B 0.000, C 0.000 }
gfCNCPoint4[24473] = {X 31.1832, Y 50.1789, Z -6.3333, A 0.000, B 0.000, C 0.000 }
gfCNCPoint4[24474] = {X 29.9993, Y 50.7716, Z -6.3333, A 0.000, B 0.000, C 0.000 }
gfCNCPoint4[24475] = {X 28.7428, Y 51.1884, Z -6.3333, A 0.000, B 0.000, C 0.000 }
gfCNCPoint4[24476] = {X 27.4394, Y 51.4208, Z -6.3333, A 0.000, B 0.000, C 0.000 }
gfCNCPoint4[24477] = {X 26.1162, Y 51.4640, Z -6.3333, A 0.000, B 0.000, C 0.000 }
gfCNCPoint4[24478] = {X 23.6773, Y 52.5826, Z -6.3333, A 0.000, B 0.000, C 0.000 }
gfCNCPoint4[24479] = {X 21.1583, Y 53.5069, Z -6.3333, A 0.000, B 0.000, C 0.000 }
gfCNCPoint4[24480] = {X 18.9468, Y 54.1360, Z -6.3333, A 0.000, B 0.000, C 0.000 }
gfCNCPoint4[24481] = {X 16.6907, Y 54.5791, Z -6.3333, A 0.000, B 0.000, C 0.000 }
gfCNCPoint4[24482] = {X 14.4056, Y 54.8331, Z -6.3333, A 0.000, B 0.000, C 0.000 }
gfCNCPoint4[24483] = {X 12.1072, Y 54.8962, Z -6.3333, A 0.000, B 0.000, C 0.000 }
gfCNCPoint4[24484] = {X 9.8116, Y 54.7680, Z -6.3333, A 0.000, B 0.000, C 0.000 }
gfCNCPoint4[24485] = {X 7.5345, Y 54.4495, Z -6.3333, A 0.000, B 0.000, C 0.000 }
gfCNCPoint4[24486] = {X 7.1093, Y 54.3684, Z -6.3333, A 0.000, B 0.000, C 0.000 }
gfCNCPoint4[24487] = {X 6.6855, Y 54.2806, Z -6.3333, A 0.000, B 0.000, C 0.000 }
gfCNCPoint4[24488] = {X 5.6883, Y 54.0443, Z -6.3333, A 0.000, B 0.000, C 0.000 }
gfCNCPoint4[24489] = {X 4.7034, Y 53.7610, Z -6.3333, A 0.000, B 0.000, C 0.000 }
gfCNCPoint4[24490] = {X 4.7034, Y 95.2951, Z -6.3333, A 0.000, B 0.000, C 0.000 }
gfCNCPoint4[24491] = {X 117.9387, Y 95.2951, Z -6.3333, A 0.000, B 0.000, C 0.000 }
gfCNCPoint4[24492] = {X 118.3607, Y 94.0795, Z -6.3333, A 0.000, B 0.000, C 0.000 }
gfCNCPoint4[24493] = {X 118.9902, Y 92.9573, Z -6.3333, A 0.000, B 0.000, C 0.000 }
gfCNCPoint4[24494] = {X 119.8075, Y 91.9634, Z -6.3333, A 0.000, B 0.000, C 0.000 }
gfCNCPoint4[24495] = {X 120.7869, Y 91.1289, Z -6.3333, A 0.000, B 0.000, C 0.000 }
gfCNCPoint4[24496] = {X 121.8980, Y 90.4799, Z -6.3333, A 0.000, B 0.000, C 0.000 }
gfCNCPoint4[24497] = {X 123.1060, Y 90.0366, Z -6.3333, A 0.000, B 0.000, C 0.000 }
gfCNCPoint4[24498] = {X 124.3732, Y 89.8130, Z -6.3333, A 0.000, B 0.000, C 0.000 }
gfCNCPoint4[24499] = {X 125.0501, Y 89.7106, Z -6.3333, A 0.000, B 0.000, C 0.000 }
gfCNCPoint4[24500] = {X 125.3582, Y 89.6646, Z -6.3333, A 0.000, B 0.000, C 0.000 }
gfCNCPoint4[24501] = {X 125.6645, Y 89.6083, Z -6.3333, A 0.000, B 0.000, C 0.000 }
gfCNCPoint4[24502] = {X 126.4927, Y 88.7965, Z -6.3333, A 0.000, B 0.000, C 0.000 }
gfCNCPoint4[24503] = {X 127.2864, Y 87.9509, Z -6.3333, A 0.000, B 0.000, C 0.000 }
gfCNCPoint4[24504] = {X 152.2074, Y 60.5842, Z -6.3333, A 0.000, B 0.000, C 0.000 }
gfCNCPoint4[24505] = {X 152.0684, Y 59.7896, Z -6.3333, A 0.000, B 0.000, C 0.000 }
gfCNCPoint4[24506] = {X 152.0181, Y 58.9845, Z -6.3333, A 0.000, B 0.000, C 0.000 }
gfCNCPoint4[24507] = {X 152.0180, Y 58.0000, Z -6.3333, A 0.000, B 0.000, C 0.000 }
gfCNCPoint4[24508] = {X 152.1286, Y 56.7358, Z -6.3333, A 0.000, B 0.000, C 0.000 }
gfCNCPoint4[24509] = {X 152.4570, Y 55.5101, Z -6.3333, A 0.000, B 0.000, C 0.000 }
gfCNCPoint4[24510] = {X 152.9933, Y 54.3600, Z -6.3333, A 0.000, B 0.000, C 0.000 }
gfCNCPoint4[24511] = {X 153.7212, Y 53.3205, Z -6.3333, A 0.000, B 0.000, C 0.000 }
gfCNCPoint4[24512] = {X 154.6185, Y 52.4232, Z -6.3333, A 0.000, B 0.000, C 0.000 }
gfCNCPoint4[24513] = {X 155.6580, Y 51.6953, Z -6.3333, A 0.000, B 0.000, C 0.000 }
gfCNCPoint4[24514] = {X 156.8081, Y 51.1590, Z -6.3333, A 0.000, B 0.000, C 0.000 }
gfCNCPoint4[24515] = {X 158.0338, Y 50.8306, Z -6.3333, A 0.000, B 0.000, C 0.000 }
gfCNCPoint4[24516] = {X 159.2980, Y 50.7200, Z -6.3333, A 0.000, B 0.000, C 0.000 }
gfCNCPoint4[24517] = {X 178.5335, Y 50.7200, Z -6.3333, A 0.000, B 0.000, C 0.000 }
gfCNCPoint4[24518] = {X 179.7876, Y 50.8288, Z -6.3333, A 0.000, B 0.000, C 0.000 }
gfCNCPoint4[24519] = {X 181.0042, Y 51.1521, Z -6.3333, A 0.000, B 0.000, C 0.000 }
gfCNCPoint4[24520] = {X 182.1470, Y 51.6801, Z -6.3333, A 0.000, B 0.000, C 0.000 }
gfCNCPoint4[24521] = {X 183.1817, Y 52.3970, Z -6.3333, A 0.000, B 0.000, C 0.000 }
gfCNCPoint4[24522] = {X 184.0893, Y 53.2955, Z -6.3333, A 0.000, B 0.000, C 0.000 }
gfCNCPoint4[24523] = {X 184.8259, Y 54.3388, Z -6.3333, A 0.000, B 0.000, C 0.000 }
gfCNCPoint4[24524] = {X 185.3689, Y 55.4948, Z -6.3333, A 0.000, B 0.000, C 0.000 }
gfCNCPoint4[24525] = {X 185.7015, Y 56.7278, Z -6.3333, A 0.000, B 0.000, C 0.000 }
gfCNCPoint4[24526] = {X 185.8135, Y 58.0000, Z -6.3333, A 0.000, B 0.000, C 0.000 }
gfCNCPoint4[24527] = {X 185.8133, Y 58.9942, Z -6.3333, A 0.000, B 0.000, C 0.000 }
gfCNCPoint4[24528] = {X 185.7648, Y 59.7746, Z -6.3333, A 0.000, B 0.000, C 0.000 }
gfCNCPoint4[24529] = {X 185.6330, Y 60.5453, Z -6.3333, A 0.000, B 0.000, C 0.000 }
gfCNCPoint4[24530] = {X 211.6621, Y 88.9547, Z -6.3333, A 0.000, B 0.000, C 0.000 }
gfCNCPoint4[24531] = {X 212.0337, Y 89.3389, Z -6.3333, A 0.000, B 0.000, C 0.000 }
gfCNCPoint4[24532] = {X 212.4255, Y 89.7024, Z -6.3333, A 0.000, B 0.000, C 0.000 }
gfCNCPoint4[24533] = {X 212.6034, Y 89.7404, Z -6.3333, A 0.000, B 0.000, C 0.000 }
gfCNCPoint4[24534] = {X 213.4474, Y 89.8467, Z -6.3333, A 0.000, B 0.000, C 0.000 }
gfCNCPoint4[24535] = {X 214.4300, Y 89.7699, Z -6.3333, A 0.000, B 0.000, C 0.000 }
gfCNCPoint4[24536] = {X 215.4141, Y 89.7161, Z -6.3333, A 0.000, B 0.000, C 0.000 }
gfCNCPoint4[24537] = {X 215.6260, Y 89.6930, Z -6.3333, A 0.000, B 0.000, C 0.000 }
gfCNCPoint4[24538] = {X 215.8206, Y 89.6063, Z -6.3333, A 0.000, B 0.000, C 0.000 }
gfCNCPoint4[24539] = {X 239.3454, Y 74.5357, Z -6.3333, A 0.000, B 0.000, C 0.000 }
gfCNCPoint4[24540] = {X 220.5438, Y 67.1577, Z -6.3333, A 0.000, B 0.000, C 0.000 }
gfCNCPoint4[24541] = {X 219.0949, Y 66.6714, Z -6.3333, A 0.000, B 0.000, C 0.000 }
gfCNCPoint4[24542] = {X 217.5999, Y 66.3541, Z -6.3333, A 0.000, B 0.000, C 0.000 }
gfCNCPoint4[24543] = {X 216.0784, Y 66.2097, Z -6.3333, A 0.000, B 0.000, C 0.000 }
gfCNCPoint4[24544] = {X 214.8518, Y 66.0622, Z -6.3333, A 0.000, B 0.000, C 0.000 }
gfCNCPoint4[24545] = {X 213.6677, Y 65.7095, Z -6.3333, A 0.000, B 0.000, C 0.000 }
gfCNCPoint4[24546] = {X 212.5604, Y 65.1616, Z -6.3333, A 0.000, B 0.000, C 0.000 }
gfCNCPoint4[24547] = {X 211.5617, Y 64.4344, Z -6.3333, A 0.000, B 0.000, C 0.000 }
gfCNCPoint4[24548] = {X 210.7003, Y 63.5488, Z -6.3333, A 0.000, B 0.000, C 0.000 }
gfCNCPoint4[24549] = {X 210.0010, Y 62.5302, Z -6.3333, A 0.000, B 0.000, C 0.000 }
gfCNCPoint4[24550] = {X 209.4841, Y 61.4081, Z -6.3333, A 0.000, B 0.000, C 0.000 }
gfCNCPoint4[24551] = {X 209.1643, Y 60.2147, Z -6.3333, A 0.000, B 0.000, C 0.000 }
gfCNCPoint4[24552] = {X 209.0510, Y 58.9845, Z -6.3333, A 0.000, B 0.000, C 0.000 }
gfCNCPoint4[24553] = {X 209.0508, Y 58.0000, Z -6.3333, A 0.000, B 0.000, C 0.000 }
gfCNCPoint4[24554] = {X 209.1477, Y 56.8162, Z -6.3333, A 0.000, B 0.000, C 0.000 }
gfCNCPoint4[24555] = {X 209.4358, Y 55.6638, Z -6.3333, A 0.000, B 0.000, C 0.000 }
gfCNCPoint4[24556] = {X 209.9075, Y 54.5737, Z -6.3333, A 0.000, B 0.000, C 0.000 }
gfCNCPoint4[24557] = {X 210.5502, Y 53.5748, Z -6.3333, A 0.000, B 0.000, C 0.000 }
gfCNCPoint4[24558] = {X 211.3467, Y 52.6937, Z -6.3333, A 0.000, B 0.000, C 0.000 }
gfCNCPoint4[24559] = {X 212.2759, Y 51.9538, Z -6.3333, A 0.000, B 0.000, C 0.000 }
gfCNCPoint4[24560] = {X 213.3131, Y 51.3749, Z -6.3333, A 0.000, B 0.000, C 0.000 }
gfCNCPoint4[24561] = {X 214.4306, Y 50.9724, Z -6.3333, A 0.000, B 0.000, C 0.000 }
gfCNCPoint4[24562] = {X 215.3724, Y 50.7834, Z -6.3333, A 0.000, B 0.000, C 0.000 }
gfCNCPoint4[24563] = {X 216.3308, Y 50.7200, Z -6.3333, A 0.000, B 0.000, C 0.000 }
gfCNCPoint4[24564] = {X 237.2617, Y 50.7200, Z -6.3333, A 0.000, B 0.000, C 0.000 }
gfCNCPoint4[24565] = {X 238.3057, Y 50.7953, Z -6.3333, A 0.000, B 0.000, C 0.000 }
gfCNCPoint4[24566] = {X 239.3282, Y 51.0195, Z -6.3333, A 0.000, B 0.000, C 0.000 }
gfCNCPoint4[24567] = {X 240.3080, Y 51.3880, Z -6.3333, A 0.000, B 0.000, C 0.000 }
gfCNCPoint4[24568] = {X 241.2247, Y 51.8932, Z -6.3333, A 0.000, B 0.000, C 0.000 }
gfCNCPoint4[24569] = {X 242.0741, Y 52.5374, Z -6.3333, A 0.000, B 0.000, C 0.000 }
gfCNCPoint4[24570] = {X 242.8202, Y 53.2988, Z -6.3333, A 0.000, B 0.000, C 0.000 }
gfCNCPoint4[24571] = {X 243.4472, Y 54.1609, Z -6.3333, A 0.000, B 0.000, C 0.000 }
gfCNCPoint4[24572] = {X 243.9415, Y 55.1054, Z -6.3333, A 0.000, B 0.000, C 0.000 }
gfCNCPoint4[24573] = {X 244.2926, Y 56.1119, Z -6.3333, A 0.000, B 0.000, C 0.000 }
gfCNCPoint4[24574] = {X 249.2039, Y 58.0271, Z -6.3333, A 0.000, B 0.000, C 0.000 }
gfCNCPoint4[24575] = {X 272.6720, Y 67.3420, Z -6.3333, A 0.000, B 0.000, C 0.000 }
gfCNCPoint4[24576] = {X 272.6719, Y 65.2838, Z -6.3333, A 0.000, B 0.000, C 0.000 }
gfCNCPoint4[24577] = {X 271.6645, Y 64.6024, Z -6.3333, A 0.000, B 0.000, C 0.000 }
gfCNCPoint4[24578] = {X 270.7846, Y 63.7628, Z -6.3333, A 0.000, B 0.000, C 0.000 }
gfCNCPoint4[24579] = {X 270.0568, Y 62.7884, Z -6.3333, A 0.000, B 0.000, C 0.000 }
gfCNCPoint4[24580] = {X 269.5013, Y 61.7065, Z -6.3333, A 0.000, B 0.000, C 0.000 }
gfCNCPoint4[24581] = {X 269.2026, Y 60.8251, Z -6.3333, A 0.000, B 0.000, C 0.000 }
gfCNCPoint4[24582] = {X 269.0188, Y 59.9128, Z -6.3333, A 0.000, B 0.000, C 0.000 }
gfCNCPoint4[24583] = {X 268.9529, Y 58.9845, Z -6.3333, A 0.000, B 0.000, C 0.000 }
gfCNCPoint4[24584] = {X 268.9527, Y 58.0000, Z -6.3333, A 0.000, B 0.000, C 0.000 }
gfCNCPoint4[24585] = {X 269.0633, Y 56.7358, Z -6.3333, A 0.000, B 0.000, C 0.000 }
gfCNCPoint4[24586] = {X 269.3917, Y 55.5101, Z -6.3333, A 0.000, B 0.000, C 0.000 }
gfCNCPoint4[24587] = {X 269.9280, Y 54.3600, Z -6.3333, A 0.000, B 0.000, C 0.000 }
gfCNCPoint4[24588] = {X 270.6559, Y 53.3205, Z -6.3333, A 0.000, B 0.000, C 0.000 }
gfCNCPoint4[24589] = {X 271.5532, Y 52.4232, Z -6.3333, A 0.000, B 0.000, C 0.000 }
gfCNCPoint4[24590] = {X 272.5927, Y 51.6953, Z -6.3333, A 0.000, B 0.000, C 0.000 }
gfCNCPoint4[24591] = {X 273.7428, Y 51.1590, Z -6.3333, A 0.000, B 0.000, C 0.000 }
gfCNCPoint4[24592] = {X 274.9685, Y 50.8306, Z -6.3333, A 0.000, B 0.000, C 0.000 }
gfCNCPoint4[24593] = {X 276.2327, Y 50.7200, Z -6.3333, A 0.000, B 0.000, C 0.000 }
gfCNCPoint4[24594] = {X 292.7731, Y 50.7200, Z -6.3333, A 0.000, B 0.000, C 0.000 }
gfCNCPoint4[24595] = {X 293.4209, Y 50.7489, Z -6.3333, A 0.000, B 0.000, C 0.000 }
gfCNCPoint4[24596] = {X 294.0636, Y 50.8353, Z -6.3333, A 0.000, B 0.000, C 0.000 }
gfCNCPoint4[24597] = {X 294.7293, Y 50.9878, Z -6.3333, A 0.000, B 0.000, C 0.000 }
gfCNCPoint4[24598] = {X 295.3778, Y 51.2019, Z -6.3333, A 0.000, B 0.000, C 0.000 }
gfCNCPoint4[24599] = {X 298.3089, Y 43.5518, Z -6.3333, A 0.000, B 0.000, C 0.000 }
gfCNCPoint4[24600] = {X 298.4821, Y 42.5288, Z -6.3333, A 0.000, B 0.000, C 0.000 }
gfCNCPoint4[24601] = {X 298.7924, Y 41.5388, Z -6.3333, A 0.000, B 0.000, C 0.000 }
gfCNCPoint4[24602] = {X 299.2341, Y 40.6000, Z -6.3333, A 0.000, B 0.000, C 0.000 }
gfCNCPoint4[24603] = {X 299.7991, Y 39.7298, Z -6.3333, A 0.000, B 0.000, C 0.000 }
gfCNCPoint4[24604] = {X 299.7991, Y 36.9943, Z -6.3333, A 0.000, B 0.000, C 0.000 }
gfCNCPoint4[24605] = {X 296.8147, Y 36.9943, Z -6.3333, A 0.000, B 0.000, C 0.000 }
gfCNCPoint4[24606] = {X 296.8144, Y 39.7482, Z -6.3333, A 0.000, B 0.000, C 0.000 }
gfCNCPoint4[24607] = {X 297.3855, Y 40.6106, Z -6.3333, A 0.000, B 0.000, C 0.000 }
gfCNCPoint4[24608] = {X 297.8304, Y 41.5444, Z -6.3333, A 0.000, B 0.000, C 0.000 }
gfCNCPoint4[24609] = {X 298.1402, Y 42.5313, Z -6.3333, A 0.000, B 0.000, C 0.000 }
gfCNCPoint4[24610] = {X 298.3089, Y 43.5518, Z -6.3333, A 0.000, B 0.000, C 0.000 }
gfCNCPoint4[24611] = {X 296.2365, Y 48.9608, Z -6.3333, A 0.000, B 0.000, C 0.000 }
gfCNCPoint4[24612] = {X 296.6125, Y 49.1140, Z -6.3333, A 0.000, B 0.000, C 0.000 }
gfCNCPoint4[24613] = {X 296.9817, Y 49.2828, Z -6.3333, A 0.000, B 0.000, C 0.000 }
gfCNCPoint4[24614] = {X 297.2571, Y 49.4212, Z -6.3333, A 0.000, B 0.000, C 0.000 }
gfCNCPoint4[24615] = {X 297.5280, Y 49.5683, Z -6.3333, A 0.000, B 0.000, C 0.000 }
gfCNCPoint4[24616] = {X 298.7174, Y 50.3602, Z -6.3333, A 0.000, B 0.000, C 0.000 }
gfCNCPoint4[24617] = {X 299.7774, Y 51.3185, Z -6.3333, A 0.000, B 0.000, C 0.000 }
gfCNCPoint4[24618] = {X 300.6847, Y 52.4224, Z -6.3333, A 0.000, B 0.000, C 0.000 }
gfCNCPoint4[24619] = {X 301.5914, Y 51.3191, Z -6.3333, A 0.000, B 0.000, C 0.000 }
gfCNCPoint4[24620] = {X 302.6506, Y 50.3611, Z -6.3333, A 0.000, B 0.000, C 0.000 }
gfCNCPoint4[24621] = {X 303.8393, Y 49.5695, Z -6.3333, A 0.000, B 0.000, C 0.000 }
gfCNCPoint4[24622] = {X 302.8989, Y 49.0956, Z -6.3333, A 0.000, B 0.000, C 0.000 }
gfCNCPoint4[24623] = {X 302.0820, Y 48.4310, Z -6.3333, A 0.000, B 0.000, C 0.000 }
gfCNCPoint4[24624] = {X 301.4268, Y 47.6067, Z -6.3333, A 0.000, B 0.000, C 0.000 }
gfCNCPoint4[24625] = {X 300.9636, Y 46.6610, Z -6.3333, A 0.000, B 0.000, C 0.000 }
gfCNCPoint4[24626] = {X 300.7923, Y 46.0759, Z -6.3333, A 0.000, B 0.000, C 0.000 }
gfCNCPoint4[24627] = {X 300.6953, Y 45.4741, Z -6.3333, A 0.000, B 0.000, C 0.000 }
gfCNCPoint4[24628] = {X 300.6790, Y 45.2570, Z -6.3333, A 0.000, B 0.000, C 0.000 }
gfCNCPoint4[24629] = {X 300.6724, Y 45.0393, Z -6.3333, A 0.000, B 0.000, C 0.000 }
gfCNCPoint4[24630] = {X 300.6725, Y 44.1882, Z -6.3333, A 0.000, B 0.000, C 0.000 }
gfCNCPoint4[24631] = {X 300.6810, Y 43.9892, Z -6.3333, A 0.000, B 0.000, C 0.000 }
gfCNCPoint4[24632] = {X 300.6970, Y 43.7906, Z -6.3333, A 0.000, B 0.000, C 0.000 }
gfCNCPoint4[24633] = {X 300.8617, Y 42.9116, Z -6.3333, A 0.000, B 0.000, C 0.000 }
gfCNCPoint4[24634] = {X 301.1737, Y 42.0735, Z -6.3333, A 0.000, B 0.000, C 0.000 }
gfCNCPoint4[24635] = {X 301.6239, Y 41.3008, Z -6.3333, A 0.000, B 0.000, C 0.000 }
gfCNCPoint4[24636] = {X 302.1991, Y 40.6160, Z -6.3333, A 0.000, B 0.000, C 0.000 }
gfCNCPoint4[24637] = {X 302.1991, Y 34.5943, Z -6.3333, A 0.000, B 0.000, C 0.000 }
gfCNCPoint4[24638] = {X 294.4149, Y 34.5943, Z -6.3333, A 0.000, B 0.000, C 0.000 }
gfCNCPoint4[24639] = {X 294.4143, Y 40.6551, Z -6.3333, A 0.000, B 0.000, C 0.000 }
gfCNCPoint4[24640] = {X 294.9944, Y 41.3218, Z -6.3333, A 0.000, B 0.000, C 0.000 }
gfCNCPoint4[24641] = {X 295.4474, Y 42.0805, Z -6.3333, A 0.000, B 0.000, C 0.000 }
gfCNCPoint4[24642] = {X 295.7590, Y 42.9073, Z -6.3333, A 0.000, B 0.000, C 0.000 }
gfCNCPoint4[24643] = {X 295.9194, Y 43.7763, Z -6.3333, A 0.000, B 0.000, C 0.000 }
gfCNCPoint4[24644] = {X 295.9350, Y 43.9923, Z -6.3333, A 0.000, B 0.000, C 0.000 }
gfCNCPoint4[24645] = {X 295.9411, Y 44.2089, Z -6.3333, A 0.000, B 0.000, C 0.000 }
gfCNCPoint4[24646] = {X 295.9411, Y 45.0000, Z -6.3333, A 0.000, B 0.000, C 0.000 }
gfCNCPoint4[24647] = {X 295.9354, Y 45.2373, Z -6.3333, A 0.000, B 0.000, C 0.000 }
gfCNCPoint4[24648] = {X 295.9180, Y 45.4741, Z -6.3333, A 0.000, B 0.000, C 0.000 }
gfCNCPoint4[24649] = {X 298.3067, Y 45.7073, Z -6.3333, A 0.000, B 0.000, C 0.000 }
gfCNCPoint4[24650] = {X 298.2010, Y 46.4214, Z -6.3333, A 0.000, B 0.000, C 0.000 }
gfCNCPoint4[24651] = {X 298.0252, Y 47.1215, Z -6.3333, A 0.000, B 0.000, C 0.000 }
gfCNCPoint4[24652] = {X 298.3689, Y 47.2942, Z -6.3333, A 0.000, B 0.000, C 0.000 }
gfCNCPoint4[24653] = {X 298.7069, Y 47.4778, Z -6.3333, A 0.000, B 0.000, C 0.000 }
gfCNCPoint4[24654] = {X 298.4514, Y 46.6051, Z -6.3333, A 0.000, B 0.000, C 0.000 }
gfCNCPoint4[24655] = {X 298.3067, Y 45.7073, Z -6.3333, A 0.000, B 0.000, C 0.000 }
gfCNCPoint4[24656] = {X 295.9180, Y 45.4741, Z -6.3333, A 0.000, B 0.000, C 0.000 }
gfCNCPoint4[24657] = {X 295.8472, Y 45.9528, Z -6.3333, A 0.000, B 0.000, C 0.000 }
gfCNCPoint4[24658] = {X 295.7293, Y 46.4221, Z -6.3333, A 0.000, B 0.000, C 0.000 }
gfCNCPoint4[24659] = {X 295.4314, Y 47.1714, Z -6.3333, A 0.000, B 0.000, C 0.000 }
gfCNCPoint4[24660] = {X 295.0142, Y 47.8614, Z -6.3333, A 0.000, B 0.000, C 0.000 }
gfCNCPoint4[24661] = {X 294.4890, Y 48.4733, Z -6.3333, A 0.000, B 0.000, C 0.000 }
gfCNCPoint4[24662] = {X 295.3742, Y 48.6760, Z -6.3333, A 0.000, B 0.000, C 0.000 }
gfCNCPoint4[24663] = {X 296.2365, Y 48.9608, Z -6.3333, A 0.000, B 0.000, C 0.000 }
gfCNCPoint4[24664] = {X 295.3778, Y 51.2019, Z -6.3333, A 0.000, B 0.000, C 0.000 }
gfCNCPoint4[24665] = {X 296.3499, Y 51.6593, Z -6.3333, A 0.000, B 0.000, C 0.000 }
gfCNCPoint4[24666] = {X 297.2441, Y 52.2547, Z -6.3333, A 0.000, B 0.000, C 0.000 }
gfCNCPoint4[24667] = {X 298.0410, Y 52.9753, Z -6.3333, A 0.000, B 0.000, C 0.000 }
gfCNCPoint4[24668] = {X 298.7231, Y 53.8053, Z -6.3333, A 0.000, B 0.000, C 0.000 }
gfCNCPoint4[24669] = {X 299.2946, Y 54.7645, Z -6.3333, A 0.000, B 0.000, C 0.000 }
gfCNCPoint4[24670] = {X 299.7126, Y 55.7997, Z -6.3333, A 0.000, B 0.000, C 0.000 }
gfCNCPoint4[24671] = {X 299.9675, Y 56.8868, Z -6.3333, A 0.000, B 0.000, C 0.000 }
gfCNCPoint4[24672] = {X 300.0531, Y 58.0000, Z -6.3333, A 0.000, B 0.000, C 0.000 }
gfCNCPoint4[24673] = {X 300.0531, Y 58.9434, Z -6.3333, A 0.000, B 0.000, C 0.000 }
gfCNCPoint4[24674] = {X 299.9649, Y 60.0535, Z -6.3333, A 0.000, B 0.000, C 0.000 }
gfCNCPoint4[24675] = {X 299.7089, Y 61.1372, Z -6.3333, A 0.000, B 0.000, C 0.000 }
gfCNCPoint4[24676] = {X 299.2909, Y 62.1693, Z -6.3333, A 0.000, B 0.000, C 0.000 }
gfCNCPoint4[24677] = {X 298.7207, Y 63.1258, Z -6.3333, A 0.000, B 0.000, C 0.000 }
gfCNCPoint4[24678] = {X 300.6824, Y 64.5085, Z -6.3333, A 0.000, B 0.000, C 0.000 }
gfCNCPoint4[24679] = {X 299.7830, Y 65.6046, Z -6.3333, A 0.000, B 0.000, C 0.000 }
gfCNCPoint4[24680] = {X 298.7334, Y 66.5578, Z -6.3333, A 0.000, B 0.000, C 0.000 }
gfCNCPoint4[24681] = {X 298.7334, Y 89.4418, Z -6.3333, A 0.000, B 0.000, C 0.000 }
gfCNCPoint4[24682] = {X 299.8301, Y 90.4463, Z -6.3333, A 0.000, B 0.000, C 0.000 }
gfCNCPoint4[24683] = {X 300.7605, Y 91.6065, Z -6.3333, A 0.000, B 0.000, C 0.000 }
gfCNCPoint4[24684] = {X 301.5029, Y 92.8951, Z -6.3333, A 0.000, B 0.000, C 0.000 }
gfCNCPoint4[24685] = {X 304.0668, Y 92.8951, Z -6.3333, A 0.000, B 0.000, C 0.000 }
gfCNCPoint4[24686] = {X 303.7093, Y 91.9007, Z -6.3333, A 0.000, B 0.000, C 0.000 }
gfCNCPoint4[24687] = {X 303.4132, Y 90.8862, Z -6.3333, A 0.000, B 0.000, C 0.000 }
gfCNCPoint4[24688] = {X 302.9739, Y 88.8153, Z -6.3333, A 0.000, B 0.000, C 0.000 }
gfCNCPoint4[24689] = {X 302.7138, Y 86.7144, Z -6.3333, A 0.000, B 0.000, C 0.000 }
gfCNCPoint4[24690] = {X 302.6347, Y 84.5988, Z -6.3333, A 0.000, B 0.000, C 0.000 }
gfCNCPoint4[24691] = {X 302.6358, Y 66.5613, Z -6.3333, A 0.000, B 0.000, C 0.000 }
gfCNCPoint4[24692] = {X 301.5836, Y 65.6068, Z -6.3333, A 0.000, B 0.000, C 0.000 }
gfCNCPoint4[24693] = {X 300.6824, Y 64.5085, Z -6.3333, A 0.000, B 0.000, C 0.000 }
gfCNCPoint4[24694] = {X 298.7207, Y 63.1258, Z -6.3333, A 0.000, B 0.000, C 0.000 }
gfCNCPoint4[24695] = {X 298.0348, Y 63.9603, Z -6.3333, A 0.000, B 0.000, C 0.000 }
gfCNCPoint4[24696] = {X 297.2331, Y 64.6843, Z -6.3333, A 0.000, B 0.000, C 0.000 }
gfCNCPoint4[24697] = {X 296.3334, Y 65.2820, Z -6.3333, A 0.000, B 0.000, C 0.000 }
gfCNCPoint4[24698] = {X 296.3334, Y 90.7160, Z -6.3333, A 0.000, B 0.000, C 0.000 }
gfCNCPoint4[24699] = {X 297.3135, Y 91.3788, Z -6.3333, A 0.000, B 0.000, C 0.000 }
gfCNCPoint4[24700] = {X 298.1739, Y 92.1910, Z -6.3333, A 0.000, B 0.000, C 0.000 }
gfCNCPoint4[24701] = {X 298.8921, Y 93.1313, Z -6.3333, A 0.000, B 0.000, C 0.000 }
gfCNCPoint4[24702] = {X 299.4492, Y 94.1751, Z -6.3333, A 0.000, B 0.000, C 0.000 }
gfCNCPoint4[24703] = {X 299.8307, Y 95.2951, Z -6.3333, A 0.000, B 0.000, C 0.000 }
gfCNCPoint4[24704] = {X 308.0989, Y 95.2951, Z -6.3333, A 0.000, B 0.000, C 0.000 }
gfCNCPoint4[24705] = {X 307.0957, Y 93.7115, Z -6.3333, A 0.000, B 0.000, C 0.000 }
gfCNCPoint4[24706] = {X 306.2994, Y 92.0145, Z -6.3333, A 0.000, B 0.000, C 0.000 }
gfCNCPoint4[24707] = {X 305.9915, Y 91.1581, Z -6.3333, A 0.000, B 0.000, C 0.000 }
gfCNCPoint4[24708] = {X 305.7365, Y 90.2845, Z -6.3333, A 0.000, B 0.000, C 0.000 }
gfCNCPoint4[24709] = {X 305.3402, Y 88.4140, Z -6.3333, A 0.000, B 0.000, C 0.000 }
gfCNCPoint4[24710] = {X 305.1056, Y 86.5165, Z -6.3333, A 0.000, B 0.000, C 0.000 }
gfCNCPoint4[24711] = {X 305.0347, Y 84.6058, Z -6.3333, A 0.000, B 0.000, C 0.000 }
gfCNCPoint4[24712] = {X 305.0358, Y 65.2840, Z -6.3333, A 0.000, B 0.000, C 0.000 }
gfCNCPoint4[24713] = {X 304.1343, Y 64.6865, Z -6.3333, A 0.000, B 0.000, C 0.000 }
gfCNCPoint4[24714] = {X 303.3313, Y 63.9619, Z -6.3333, A 0.000, B 0.000, C 0.000 }
gfCNCPoint4[24715] = {X 302.6445, Y 63.1264, Z -6.3333, A 0.000, B 0.000, C 0.000 }
gfCNCPoint4[24716] = {X 302.0794, Y 62.1789, Z -6.3333, A 0.000, B 0.000, C 0.000 }
gfCNCPoint4[24717] = {X 301.6639, Y 61.1569, Z -6.3333, A 0.000, B 0.000, C 0.000 }
gfCNCPoint4[24718] = {X 301.4076, Y 60.0839, Z -6.3333, A 0.000, B 0.000, C 0.000 }
gfCNCPoint4[24719] = {X 301.3164, Y 58.9845, Z -6.3333, A 0.000, B 0.000, C 0.000 }
gfCNCPoint4[24720] = {X 301.3162, Y 58.0000, Z -6.3333, A 0.000, B 0.000, C 0.000 }
gfCNCPoint4[24721] = {X 301.4018, Y 56.8868, Z -6.3333, A 0.000, B 0.000, C 0.000 }
gfCNCPoint4[24722] = {X 301.6567, Y 55.7997, Z -6.3333, A 0.000, B 0.000, C 0.000 }
gfCNCPoint4[24723] = {X 302.0747, Y 54.7645, Z -6.3333, A 0.000, B 0.000, C 0.000 }
gfCNCPoint4[24724] = {X 302.6462, Y 53.8053, Z -6.3333, A 0.000, B 0.000, C 0.000 }
gfCNCPoint4[24725] = {X 303.3281, Y 52.9755, Z -6.3333, A 0.000, B 0.000, C 0.000 }
gfCNCPoint4[24726] = {X 304.1247, Y 52.2551, Z -6.3333, A 0.000, B 0.000, C 0.000 }
gfCNCPoint4[24727] = {X 305.0187, Y 51.6597, Z -6.3333, A 0.000, B 0.000, C 0.000 }
gfCNCPoint4[24728] = {X 306.1514, Y 51.1428, Z -6.3333, A 0.000, B 0.000, C 0.000 }
gfCNCPoint4[24729] = {X 307.3557, Y 50.8265, Z -6.3333, A 0.000, B 0.000, C 0.000 }
gfCNCPoint4[24730] = {X 308.5962, Y 50.7200, Z -6.3333, A 0.000, B 0.000, C 0.000 }
gfCNCPoint4[24731] = {X 324.3107, Y 50.7200, Z -6.3333, A 0.000, B 0.000, C 0.000 }
gfCNCPoint4[24732] = {X 325.2469, Y 50.7804, Z -6.3333, A 0.000, B 0.000, C 0.000 }
gfCNCPoint4[24733] = {X 326.1675, Y 50.9608, Z -6.3333, A 0.000, B 0.000, C 0.000 }
gfCNCPoint4[24734] = {X 326.5260, Y 51.0653, Z -6.3333, A 0.000, B 0.000, C 0.000 }
gfCNCPoint4[24735] = {X 326.8787, Y 51.1880, Z -6.3333, A 0.000, B 0.000, C 0.000 }
gfCNCPoint4[24736] = {X 327.4517, Y 51.4325, Z -6.3333, A 0.000, B 0.000, C 0.000 }
gfCNCPoint4[24737] = {X 328.0017, Y 51.7251, Z -6.3333, A 0.000, B 0.000, C 0.000 }
gfCNCPoint4[24738] = {X 328.5430, Y 52.0766, Z -6.3333, A 0.000, B 0.000, C 0.000 }
gfCNCPoint4[24739] = {X 329.0510, Y 52.4748, Z -6.3333, A 0.000, B 0.000, C 0.000 }
gfCNCPoint4[24740] = {X 329.9283, Y 53.3695, Z -6.3333, A 0.000, B 0.000, C 0.000 }
gfCNCPoint4[24741] = {X 330.6391, Y 54.4015, Z -6.3333, A 0.000, B 0.000, C 0.000 }
gfCNCPoint4[24742] = {X 331.1625, Y 55.5401, Z -6.3333, A 0.000, B 0.000, C 0.000 }
gfCNCPoint4[24743] = {X 331.4828, Y 56.7515, Z -6.3333, A 0.000, B 0.000, C 0.000 }
gfCNCPoint4[24744] = {X 331.5907, Y 58.0000, Z -6.3333, A 0.000, B 0.000, C 0.000 }
gfCNCPoint4[24745] = {X 331.5907, Y 58.9394, Z -6.3333, A 0.000, B 0.000, C 0.000 }
gfCNCPoint4[24746] = {X 331.4736, Y 60.2165, Z -6.3333, A 0.000, B 0.000, C 0.000 }
gfCNCPoint4[24747] = {X 331.1353, Y 61.4535, Z -6.3333, A 0.000, B 0.000, C 0.000 }
gfCNCPoint4[24748] = {X 330.5862, Y 62.6125, Z -6.3333, A 0.000, B 0.000, C 0.000 }
gfCNCPoint4[24749] = {X 329.8433, Y 63.6578, Z -6.3333, A 0.000, B 0.000, C 0.000 }
gfCNCPoint4[24750] = {X 328.9293, Y 64.5574, Z -6.3333, A 0.000, B 0.000, C 0.000 }
gfCNCPoint4[24751] = {X 327.8723, Y 65.2836, Z -6.3333, A 0.000, B 0.000, C 0.000 }
gfCNCPoint4[24752] = {X 327.8739, Y 83.2150, Z -6.3333, A 0.000, B 0.000, C 0.000 }
gfCNCPoint4[24753] = {X 327.8874, Y 84.5913, Z -6.3333, A 0.000, B 0.000, C 0.000 }
gfCNCPoint4[24754] = {X 327.8969, Y 84.9539, Z -6.3333, A 0.000, B 0.000, C 0.000 }
gfCNCPoint4[24755] = {X 327.9238, Y 85.3156, Z -6.3333, A 0.000, B 0.000, C 0.000 }
gfCNCPoint4[24756] = {X 328.8618, Y 85.6716, Z -6.3333, A 0.000, B 0.000, C 0.000 }
gfCNCPoint4[24757] = {X 329.8278, Y 85.9424, Z -6.3333, A 0.000, B 0.000, C 0.000 }
gfCNCPoint4[24758] = {X 331.9607, Y 86.3866, Z -6.3333, A 0.000, B 0.000, C 0.000 }
gfCNCPoint4[24759] = {X 334.1129, Y 86.7254, Z -6.3333, A 0.000, B 0.000, C 0.000 }
gfCNCPoint4[24760] = {X 336.2791, Y 86.9580, Z -6.3333, A 0.000, B 0.000, C 0.000 }
gfCNCPoint4[24761] = {X 340.5610, Y 87.2463, Z -6.3333, A 0.000, B 0.000, C 0.000 }
gfCNCPoint4[24762] = {X 344.8499, Y 87.3968, Z -6.3333, A 0.000, B 0.000, C 0.000 }
gfCNCPoint4[24763] = {X 349.1414, Y 87.4094, Z -6.3333, A 0.000, B 0.000, C 0.000 }
gfCNCPoint4[24764] = {X 353.1933, Y 87.3435, Z -6.3333, A 0.000, B 0.000, C 0.000 }
gfCNCPoint4[24765] = {X 357.2401, Y 87.1303, Z -6.3333, A 0.000, B 0.000, C 0.000 }
gfCNCPoint4[24766] = {X 361.2764, Y 86.7700, Z -6.3333, A 0.000, B 0.000, C 0.000 }
gfCNCPoint4[24767] = {X 363.1972, Y 86.5048, Z -6.3333, A 0.000, B 0.000, C 0.000 }
gfCNCPoint4[24768] = {X 365.1004, Y 86.1335, Z -6.3333, A 0.000, B 0.000, C 0.000 }
gfCNCPoint4[24769] = {X 366.9800, Y 85.6571, Z -6.3333, A 0.000, B 0.000, C 0.000 }
gfCNCPoint4[24770] = {X 367.4410, Y 85.5106, Z -6.3333, A 0.000, B 0.000, C 0.000 }
gfCNCPoint4[24771] = {X 367.8882, Y 85.3262, Z -6.3333, A 0.000, B 0.000, C 0.000 }
gfCNCPoint4[24772] = {X 367.9416, Y 84.5784, Z -6.3333, A 0.000, B 0.000, C 0.000 }
gfCNCPoint4[24773] = {X 367.9594, Y 83.8288, Z -6.3333, A 0.000, B 0.000, C 0.000 }
gfCNCPoint4[24774] = {X 367.9583, Y 65.2837, Z -6.3333, A 0.000, B 0.000, C 0.000 }
gfCNCPoint4[24775] = {X 366.9045, Y 64.5646, Z -6.3333, A 0.000, B 0.000, C 0.000 }
gfCNCPoint4[24776] = {X 365.9925, Y 63.6726, Z -6.3333, A 0.000, B 0.000, C 0.000 }
gfCNCPoint4[24777] = {X 365.2502, Y 62.6351, Z -6.3333, A 0.000, B 0.000, C 0.000 }
gfCNCPoint4[24778] = {X 364.7004, Y 61.4839, Z -6.3333, A 0.000, B 0.000, C 0.000 }
gfCNCPoint4[24779] = {X 364.3600, Y 60.2545, Z -6.3333, A 0.000, B 0.000, C 0.000 }
gfCNCPoint4[24780] = {X 364.2395, Y 58.9845, Z -6.3333, A 0.000, B 0.000, C 0.000 }
gfCNCPoint4[24781] = {X 364.2393, Y 58.0000, Z -6.3333, A 0.000, B 0.000, C 0.000 }
gfCNCPoint4[24782] = {X 364.3499, Y 56.7358, Z -6.3333, A 0.000, B 0.000, C 0.000 }
gfCNCPoint4[24783] = {X 364.6783, Y 55.5101, Z -6.3333, A 0.000, B 0.000, C 0.000 }
gfCNCPoint4[24784] = {X 365.2146, Y 54.3600, Z -6.3333, A 0.000, B 0.000, C 0.000 }
gfCNCPoint4[24785] = {X 365.9425, Y 53.3205, Z -6.3333, A 0.000, B 0.000, C 0.000 }
gfCNCPoint4[24786] = {X 366.8398, Y 52.4232, Z -6.3333, A 0.000, B 0.000, C 0.000 }
gfCNCPoint4[24787] = {X 367.8793, Y 51.6953, Z -6.3333, A 0.000, B 0.000, C 0.000 }
gfCNCPoint4[24788] = {X 369.0294, Y 51.1590, Z -6.3333, A 0.000, B 0.000, C 0.000 }
gfCNCPoint4[24789] = {X 370.2551, Y 50.8306, Z -6.3333, A 0.000, B 0.000, C 0.000 }
gfCNCPoint4[24790] = {X 371.5193, Y 50.7200, Z -6.3333, A 0.000, B 0.000, C 0.000 }
gfCNCPoint4[24791] = {X 388.0597, Y 50.7200, Z -6.3333, A 0.000, B 0.000, C 0.000 }
gfCNCPoint4[24792] = {X 389.2271, Y 50.8142, Z -6.3333, A 0.000, B 0.000, C 0.000 }
gfCNCPoint4[24793] = {X 390.3643, Y 51.0944, Z -6.3333, A 0.000, B 0.000, C 0.000 }
gfCNCPoint4[24794] = {X 391.4418, Y 51.5533, Z -6.3333, A 0.000, B 0.000, C 0.000 }
gfCNCPoint4[24795] = {X 392.4319, Y 52.1791, Z -6.3333, A 0.000, B 0.000, C 0.000 }
gfCNCPoint4[24796] = {X 393.3087, Y 52.9556, Z -6.3333, A 0.000, B 0.000, C 0.000 }
gfCNCPoint4[24797] = {X 394.1855, Y 52.1791, Z -6.3333, A 0.000, B 0.000, C 0.000 }
gfCNCPoint4[24798] = {X 395.1756, Y 51.5533, Z -6.3333, A 0.000, B 0.000, C 0.000 }
gfCNCPoint4[24799] = {X 396.2531, Y 51.0944, Z -6.3333, A 0.000, B 0.000, C 0.000 }
gfCNCPoint4[24800] = {X 397.3903, Y 50.8142, Z -6.3333, A 0.000, B 0.000, C 0.000 }
gfCNCPoint4[24801] = {X 398.5577, Y 50.7200, Z -6.3333, A 0.000, B 0.000, C 0.000 }
gfCNCPoint4[24802] = {X 419.4886, Y 50.7200, Z -6.3333, A 0.000, B 0.000, C 0.000 }
gfCNCPoint4[24803] = {X 420.6739, Y 50.8171, Z -6.3333, A 0.000, B 0.000, C 0.000 }
gfCNCPoint4[24804] = {X 421.8275, Y 51.1060, Z -6.3333, A 0.000, B 0.000, C 0.000 }
gfCNCPoint4[24805] = {X 422.9188, Y 51.5788, Z -6.3333, A 0.000, B 0.000, C 0.000 }
gfCNCPoint4[24806] = {X 423.9185, Y 52.2229, Z -6.3333, A 0.000, B 0.000, C 0.000 }
gfCNCPoint4[24807] = {X 424.8000, Y 53.0213, Z -6.3333, A 0.000, B 0.000, C 0.000 }
gfCNCPoint4[24808] = {X 425.5397, Y 53.9525, Z -6.3333, A 0.000, B 0.000, C 0.000 }
gfCNCPoint4[24809] = {X 426.1180, Y 54.9917, Z -6.3333, A 0.000, B 0.000, C 0.000 }
gfCNCPoint4[24810] = {X 426.5193, Y 56.1112, Z -6.3333, A 0.000, B 0.000, C 0.000 }
gfCNCPoint4[24811] = {X 430.7007, Y 57.7403, Z -6.3333, A 0.000, B 0.000, C 0.000 }
gfCNCPoint4[24812] = {X 454.8984, Y 67.3412, Z -6.3333, A 0.000, B 0.000, C 0.000 }
gfCNCPoint4[24813] = {X 454.8985, Y 65.2836, Z -6.3333, A 0.000, B 0.000, C 0.000 }
gfCNCPoint4[24814] = {X 453.8913, Y 64.6023, Z -6.3333, A 0.000, B 0.000, C 0.000 }
gfCNCPoint4[24815] = {X 453.0115, Y 63.7628, Z -6.3333, A 0.000, B 0.000, C 0.000 }
gfCNCPoint4[24816] = {X 452.2838, Y 62.7886, Z -6.3333, A 0.000, B 0.000, C 0.000 }
gfCNCPoint4[24817] = {X 451.7283, Y 61.7069, Z -6.3333, A 0.000, B 0.000, C 0.000 }
gfCNCPoint4[24818] = {X 451.4296, Y 60.8253, Z -6.3333, A 0.000, B 0.000, C 0.000 }
gfCNCPoint4[24819] = {X 451.2457, Y 59.9129, Z -6.3333, A 0.000, B 0.000, C 0.000 }
gfCNCPoint4[24820] = {X 451.1798, Y 58.9845, Z -6.3333, A 0.000, B 0.000, C 0.000 }
gfCNCPoint4[24821] = {X 451.1796, Y 58.0000, Z -6.3333, A 0.000, B 0.000, C 0.000 }
gfCNCPoint4[24822] = {X 451.2795, Y 56.7981, Z -6.3333, A 0.000, B 0.000, C 0.000 }
gfCNCPoint4[24823] = {X 451.5765, Y 55.6291, Z -6.3333, A 0.000, B 0.000, C 0.000 }
gfCNCPoint4[24824] = {X 452.0624, Y 54.5253, Z -6.3333, A 0.000, B 0.000, C 0.000 }
gfCNCPoint4[24825] = {X 452.7238, Y 53.5168, Z -6.3333, A 0.000, B 0.000, C 0.000 }
gfCNCPoint4[24826] = {X 453.5427, Y 52.6313, Z -6.3333, A 0.000, B 0.000, C 0.000 }
gfCNCPoint4[24827] = {X 454.4966, Y 51.8932, Z -6.3333, A 0.000, B 0.000, C 0.000 }
gfCNCPoint4[24828] = {X 455.4133, Y 51.3880, Z -6.3333, A 0.000, B 0.000, C 0.000 }
gfCNCPoint4[24829] = {X 456.3931, Y 51.0195, Z -6.3333, A 0.000, B 0.000, C 0.000 }
gfCNCPoint4[24830] = {X 457.4155, Y 50.7953, Z -6.3333, A 0.000, B 0.000, C 0.000 }
gfCNCPoint4[24831] = {X 458.4596, Y 50.7200, Z -6.3333, A 0.000, B 0.000, C 0.000 }
gfCNCPoint4[24832] = {X 475.0000, Y 50.7200, Z -6.3333, A 0.000, B 0.000, C 0.000 }
gfCNCPoint4[24833] = {X 476.0441, Y 50.7953, Z -6.3333, A 0.000, B 0.000, C 0.000 }
gfCNCPoint4[24834] = {X 477.0665, Y 51.0195, Z -6.3333, A 0.000, B 0.000, C 0.000 }
gfCNCPoint4[24835] = {X 478.0463, Y 51.3880, Z -6.3333, A 0.000, B 0.000, C 0.000 }
gfCNCPoint4[24836] = {X 478.9630, Y 51.8932, Z -6.3333, A 0.000, B 0.000, C 0.000 }
gfCNCPoint4[24837] = {X 479.9169, Y 52.6313, Z -6.3333, A 0.000, B 0.000, C 0.000 }
gfCNCPoint4[24838] = {X 480.7358, Y 53.5168, Z -6.3333, A 0.000, B 0.000, C 0.000 }
gfCNCPoint4[24839] = {X 481.3972, Y 54.5253, Z -6.3333, A 0.000, B 0.000, C 0.000 }
gfCNCPoint4[24840] = {X 481.8831, Y 55.6291, Z -6.3333, A 0.000, B 0.000, C 0.000 }
gfCNCPoint4[24841] = {X 482.1801, Y 56.7981, Z -6.3333, A 0.000, B 0.000, C 0.000 }
gfCNCPoint4[24842] = {X 482.2800, Y 58.0000, Z -6.3333, A 0.000, B 0.000, C 0.000 }
gfCNCPoint4[24843] = {X 482.2798, Y 58.9942, Z -6.3333, A 0.000, B 0.000, C 0.000 }
gfCNCPoint4[24844] = {X 482.1578, Y 60.2625, Z -6.3333, A 0.000, B 0.000, C 0.000 }
gfCNCPoint4[24845] = {X 481.8165, Y 61.4901, Z -6.3333, A 0.000, B 0.000, C 0.000 }
gfCNCPoint4[24846] = {X 481.2665, Y 62.6394, Z -6.3333, A 0.000, B 0.000, C 0.000 }
gfCNCPoint4[24847] = {X 480.5245, Y 63.6752, Z -6.3333, A 0.000, B 0.000, C 0.000 }
gfCNCPoint4[24848] = {X 479.6133, Y 64.5658, Z -6.3333, A 0.000, B 0.000, C 0.000 }
gfCNCPoint4[24849] = {X 478.5608, Y 65.2838, Z -6.3333, A 0.000, B 0.000, C 0.000 }
gfCNCPoint4[24850] = {X 478.5612, Y 90.7247, Z -6.3333, A 0.000, B 0.000, C 0.000 }
gfCNCPoint4[24851] = {X 479.5432, Y 91.3836, Z -6.3333, A 0.000, B 0.000, C 0.000 }
gfCNCPoint4[24852] = {X 480.4052, Y 92.1932, Z -6.3333, A 0.000, B 0.000, C 0.000 }
gfCNCPoint4[24853] = {X 481.1243, Y 93.1321, Z -6.3333, A 0.000, B 0.000, C 0.000 }
gfCNCPoint4[24854] = {X 481.6814, Y 94.1753, Z -6.3333, A 0.000, B 0.000, C 0.000 }
gfCNCPoint4[24855] = {X 482.0617, Y 95.2951, Z -6.3333, A 0.000, B 0.000, C 0.000 }
gfCNCPoint4[24856] = {X 507.6813, Y 95.2951, Z -6.3333, A 0.000, B 0.000, C 0.000 }
gfCNCPoint4[24857] = {X 507.6813, Y 97.6951, Z -6.3333, A 0.000, B 0.000, C 0.000 }
gfCNCPoint4[24858] = {X 597.6966, Y 97.6951, Z -6.3333, A 0.000, B 0.000, C 0.000 }
gfCNCPoint4[24859] = {X 597.6966, Y 51.8000, Z -6.3333, A 0.000, B 0.000, C 0.000 }
gfCNCPoint4[24860] = {X 593.5565, Y 51.8000, Z -6.3333, A 0.000, B 0.000, C 0.000 }
gfCNCPoint4[24861] = {X 592.3428, Y 51.6908, Z -6.3333, A 0.000, B 0.000, C 0.000 }
gfCNCPoint4[24862] = {X 591.1680, Y 51.3667, Z -6.3333, A 0.000, B 0.000, C 0.000 }
gfCNCPoint4[24863] = {X 590.0699, Y 50.8381, Z -6.3333, A 0.000, B 0.000, C 0.000 }
gfCNCPoint4[24864] = {X 589.0838, Y 50.1220, Z -6.3333, A 0.000, B 0.000, C 0.000 }
gfCNCPoint4[24865] = {X 588.4736, Y 49.5171, Z -6.3333, A 0.000, B 0.000, C 0.000 }
gfCNCPoint4[24866] = {X 587.9446, Y 48.8401, Z -6.3333, A 0.000, B 0.000, C 0.000 }
gfCNCPoint4[24867] = {X 587.5052, Y 48.1018, Z -6.3333, A 0.000, B 0.000, C 0.000 }
gfCNCPoint4[24868] = {X 587.0658, Y 48.8401, Z -6.3333, A 0.000, B 0.000, C 0.000 }
gfCNCPoint4[24869] = {X 586.5368, Y 49.5171, Z -6.3333, A 0.000, B 0.000, C 0.000 }
gfCNCPoint4[24870] = {X 585.9266, Y 50.1220, Z -6.3333, A 0.000, B 0.000, C 0.000 }
gfCNCPoint4[24871] = {X 585.1803, Y 50.6880, Z -6.3333, A 0.000, B 0.000, C 0.000 }
gfCNCPoint4[24872] = {X 584.3634, Y 51.1461, Z -6.3333, A 0.000, B 0.000, C 0.000 }
gfCNCPoint4[24873] = {X 583.3013, Y 51.5442, Z -6.3333, A 0.000, B 0.000, C 0.000 }
gfCNCPoint4[24874] = {X 582.1877, Y 51.7603, Z -6.3333, A 0.000, B 0.000, C 0.000 }
gfCNCPoint4[24875] = {X 581.0538, Y 51.7882, Z -6.3333, A 0.000, B 0.000, C 0.000 }
gfCNCPoint4[24876] = {X 579.9310, Y 51.6273, Z -6.3333, A 0.000, B 0.000, C 0.000 }
gfCNCPoint4[24877] = {X 578.8505, Y 51.2819, Z -6.3333, A 0.000, B 0.000, C 0.000 }
gfCNCPoint4[24878] = {X 577.8425, Y 50.7618, Z -6.3333, A 0.000, B 0.000, C 0.000 }
gfCNCPoint4[24879] = {X 576.9350, Y 50.0813, Z -6.3333, A 0.000, B 0.000, C 0.000 }
gfCNCPoint4[24880] = {X 576.3133, Y 49.4513, Z -6.3333, A 0.000, B 0.000, C 0.000 }
gfCNCPoint4[24881] = {X 575.7786, Y 48.7459, Z -6.3333, A 0.000, B 0.000, C 0.000 }
gfCNCPoint4[24882] = {X 575.3401, Y 47.9770, Z -6.3333, A 0.000, B 0.000, C 0.000 }
gfCNCPoint4[24883] = {X 574.7637, Y 48.9470, Z -6.3333, A 0.000, B 0.000, C 0.000 }
gfCNCPoint4[24884] = {X 574.0348, Y 49.8083, Z -6.3333, A 0.000, B 0.000, C 0.000 }
gfCNCPoint4[24885] = {X 573.8920, Y 49.9470, Z -6.3333, A 0.000, B 0.000, C 0.000 }
gfCNCPoint4[24886] = {X 573.7453, Y 50.0813, Z -6.3333, A 0.000, B 0.000, C 0.000 }
gfCNCPoint4[24887] = {X 572.7526, Y 50.8143, Z -6.3333, A 0.000, B 0.000, C 0.000 }
gfCNCPoint4[24888] = {X 571.6437, Y 51.3558, Z -6.3333, A 0.000, B 0.000, C 0.000 }
gfCNCPoint4[24889] = {X 570.4553, Y 51.6880, Z -6.3333, A 0.000, B 0.000, C 0.000 }
gfCNCPoint4[24890] = {X 569.2264, Y 51.8000, Z -6.3333, A 0.000, B 0.000, C 0.000 }
gfCNCPoint4[24891] = {X 562.4443, Y 51.8000, Z -6.3333, A 0.000, B 0.000, C 0.000 }
gfCNCPoint4[24892] = {X 561.2348, Y 51.6916, Z -6.3333, A 0.000, B 0.000, C 0.000 }
gfCNCPoint4[24893] = {X 560.0638, Y 51.3697, Z -6.3333, A 0.000, B 0.000, C 0.000 }
gfCNCPoint4[24894] = {X 558.9688, Y 50.8447, Z -6.3333, A 0.000, B 0.000, C 0.000 }
gfCNCPoint4[24895] = {X 557.9846, Y 50.1333, Z -6.3333, A 0.000, B 0.000, C 0.000 }
gfCNCPoint4[24896] = {X 557.1757, Y 49.2990, Z -6.3333, A 0.000, B 0.000, C 0.000 }
gfCNCPoint4[24897] = {X 556.5206, Y 48.3392, Z -6.3333, A 0.000, B 0.000, C 0.000 }
gfCNCPoint4[24898] = {X 556.0386, Y 47.2818, Z -6.3333, A 0.000, B 0.000, C 0.000 }
gfCNCPoint4[24899] = {X 555.7436, Y 46.1578, Z -6.3333, A 0.000, B 0.000, C 0.000 }
gfCNCPoint4[24900] = {X 555.6443, Y 45.0000, Z -6.3333, A 0.000, B 0.000, C 0.000 }
gfCNCPoint4[24901] = {X 555.6443, Y 44.0558, Z -6.3333, A 0.000, B 0.000, C 0.000 }
gfCNCPoint4[24902] = {X 555.7464, Y 42.9037, Z -6.3333, A 0.000, B 0.000, C 0.000 }
gfCNCPoint4[24903] = {X 556.0414, Y 41.7852, Z -6.3333, A 0.000, B 0.000, C 0.000 }
gfCNCPoint4[24904] = {X 556.5209, Y 40.7326, Z -6.3333, A 0.000, B 0.000, C 0.000 }
gfCNCPoint4[24905] = {X 557.1712, Y 39.7760, Z -6.3333, A 0.000, B 0.000, C 0.000 }
gfCNCPoint4[24906] = {X 557.1712, Y 10.2276, Z -6.3333, A 0.000, B 0.000, C 0.000 }
gfCNCPoint4[24907] = {X 556.5253, Y 9.2815, Z -6.3333, A 0.000, B 0.000, C 0.000 }
gfCNCPoint4[24908] = {X 556.0474, Y 8.2405, Z -6.3333, A 0.000, B 0.000, C 0.000 }
gfCNCPoint4[24909] = {X 555.7510, Y 7.1340, Z -6.3333, A 0.000, B 0.000, C 0.000 }
gfCNCPoint4[24910] = {X 555.6446, Y 5.9935, Z -6.3333, A 0.000, B 0.000, C 0.000 }
gfCNCPoint4[24911] = {X 555.6443, Y 5.0000, Z -6.3333, A 0.000, B 0.000, C 0.000 }
gfCNCPoint4[24912] = {X 555.6452, Y 4.8909, Z -6.3333, A 0.000, B 0.000, C 0.000 }
gfCNCPoint4[24913] = {X 555.6478, Y 4.7819, Z -6.3333, A 0.000, B 0.000, C 0.000 }
gfCNCPoint4[24914] = {X 555.8079, Y 3.5173, Z -6.3333, A 0.000, B 0.000, C 0.000 }
gfCNCPoint4[24915] = {X 556.2012, Y 2.3049, Z -6.3333, A 0.000, B 0.000, C 0.000 }
gfCNCPoint4[24916] = {X 358.2605, Y 2.3049, Z -6.3333, A 0.000, B 0.000, C 0.000 }
gfCNCPoint4[24917] = {X 360.1216, Y 3.4745, Z -6.3333, A 0.000, B 0.000, C 0.000 }
gfCNCPoint4[24918] = {X 361.8541, Y 4.8273, Z -6.3333, A 0.000, B 0.000, C 0.000 }
gfCNCPoint4[24919] = {X 363.4400, Y 6.3495, Z -6.3333, A 0.000, B 0.000, C 0.000 }
gfCNCPoint4[24920] = {X 363.8251, Y 6.7699, Z -6.3333, A 0.000, B 0.000, C 0.000 }
gfCNCPoint4[24921] = {X 364.1991, Y 7.2003, Z -6.3333, A 0.000, B 0.000, C 0.000 }
gfCNCPoint4[24922] = {X 365.5804, Y 8.9957, Z -6.3333, A 0.000, B 0.000, C 0.000 }
gfCNCPoint4[24923] = {X 366.7980, Y 10.9059, Z -6.3333, A 0.000, B 0.000, C 0.000 }
gfCNCPoint4[24924] = {X 367.8424, Y 12.9160, Z -6.3333, A 0.000, B 0.000, C 0.000 }
gfCNCPoint4[24925] = {X 368.7055, Y 15.0104, Z -6.3333, A 0.000, B 0.000, C 0.000 }
gfCNCPoint4[24926] = {X 369.3805, Y 17.1728, Z -6.3333, A 0.000, B 0.000, C 0.000 }
gfCNCPoint4[24927] = {X 369.8622, Y 19.3862, Z -6.3333, A 0.000, B 0.000, C 0.000 }
gfCNCPoint4[24928] = {X 370.1988, Y 21.7960, Z -6.3333, A 0.000, B 0.000, C 0.000 }
gfCNCPoint4[24929] = {X 370.3531, Y 24.2243, Z -6.3333, A 0.000, B 0.000, C 0.000 }
gfCNCPoint4[24930] = {X 370.3242, Y 26.6574, Z -6.3333, A 0.000, B 0.000, C 0.000 }
gfCNCPoint4[24931] = {X 370.1123, Y 29.0813, Z -6.3333, A 0.000, B 0.000, C 0.000 }
gfCNCPoint4[24932] = {X 369.7185, Y 31.4824, Z -6.3333, A 0.000, B 0.000, C 0.000 }
gfCNCPoint4[24933] = {X 369.1827, Y 33.6341, Z -6.3333, A 0.000, B 0.000, C 0.000 }
gfCNCPoint4[24934] = {X 368.4590, Y 35.7301, Z -6.3333, A 0.000, B 0.000, C 0.000 }
gfCNCPoint4[24935] = {X 367.5530, Y 37.7540, Z -6.3333, A 0.000, B 0.000, C 0.000 }
gfCNCPoint4[24936] = {X 366.4720, Y 39.6900, Z -6.3333, A 0.000, B 0.000, C 0.000 }
gfCNCPoint4[24937] = {X 365.2242, Y 41.5230, Z -6.3333, A 0.000, B 0.000, C 0.000 }
gfCNCPoint4[24938] = {X 365.1115, Y 41.6772, Z -6.3333, A 0.000, B 0.000, C 0.000 }
gfCNCPoint4[24939] = {X 363.6769, Y 43.3969, Z -6.3333, A 0.000, B 0.000, C 0.000 }
gfCNCPoint4[24940] = {X 362.0787, Y 44.9658, Z -6.3333, A 0.000, B 0.000, C 0.000 }
gfCNCPoint4[24941] = {X 360.3328, Y 46.3683, Z -6.3333, A 0.000, B 0.000, C 0.000 }
gfCNCPoint4[24942] = {X 358.4563, Y 47.5907, Z -6.3333, A 0.000, B 0.000, C 0.000 }
gfCNCPoint4[24943] = {X 356.4678, Y 48.6209, Z -6.3333, A 0.000, B 0.000, C 0.000 }
gfCNCPoint4[24944] = {X 354.6708, Y 49.3149, Z -6.3333, A 0.000, B 0.000, C 0.000 }
gfCNCPoint4[24945] = {X 352.8231, Y 49.8598, Z -6.3333, A 0.000, B 0.000, C 0.000 }
gfCNCPoint4[24946] = {X 350.9372, Y 50.2521, Z -6.3333, A 0.000, B 0.000, C 0.000 }
gfCNCPoint4[24947] = {X 349.0255, Y 50.4893, Z -6.3333, A 0.000, B 0.000, C 0.000 }
gfCNCPoint4[24948] = {X 347.1008, Y 50.5696, Z -6.3333, A 0.000, B 0.000, C 0.000 }
gfCNCPoint4[24949] = {X 344.9874, Y 50.5334, Z -6.3333, A 0.000, B 0.000, C 0.000 }
gfCNCPoint4[24950] = {X 342.8850, Y 50.3141, Z -6.3333, A 0.000, B 0.000, C 0.000 }
gfCNCPoint4[24951] = {X 340.8096, Y 49.9135, Z -6.3333, A 0.000, B 0.000, C 0.000 }
gfCNCPoint4[24952] = {X 338.7767, Y 49.3346, Z -6.3333, A 0.000, B 0.000, C 0.000 }
gfCNCPoint4[24953] = {X 336.8016, Y 48.5817, Z -6.3333, A 0.000, B 0.000, C 0.000 }
gfCNCPoint4[24954] = {X 334.8992, Y 47.6605, Z -6.3333, A 0.000, B 0.000, C 0.000 }
gfCNCPoint4[24955] = {X 333.3422, Y 46.7035, Z -6.3333, A 0.000, B 0.000, C 0.000 }
gfCNCPoint4[24956] = {X 331.8610, Y 45.6330, Z -6.3333, A 0.000, B 0.000, C 0.000 }
gfCNCPoint4[24957] = {X 330.4639, Y 44.4550, Z -6.3333, A 0.000, B 0.000, C 0.000 }
gfCNCPoint4[24958] = {X 329.4666, Y 44.4079, Z -6.3333, A 0.000, B 0.000, C 0.000 }
gfCNCPoint4[24959] = {X 328.4998, Y 44.1588, Z -6.3333, A 0.000, B 0.000, C 0.000 }
gfCNCPoint4[24960] = {X 327.6038, Y 43.7181, Z -6.3333, A 0.000, B 0.000, C 0.000 }
gfCNCPoint4[24961] = {X 326.8164, Y 43.1044, Z -6.3333, A 0.000, B 0.000, C 0.000 }
gfCNCPoint4[24962] = {X 326.1897, Y 42.4934, Z -6.3333, A 0.000, B 0.000, C 0.000 }
gfCNCPoint4[24963] = {X 325.5686, Y 41.7541, Z -6.3333, A 0.000, B 0.000, C 0.000 }
gfCNCPoint4[24964] = {X 325.1052, Y 40.9070, Z -6.3333, A 0.000, B 0.000, C 0.000 }
gfCNCPoint4[24965] = {X 324.8177, Y 39.9852, Z -6.3333, A 0.000, B 0.000, C 0.000 }
gfCNCPoint4[24966] = {X 324.7172, Y 39.0249, Z -6.3333, A 0.000, B 0.000, C 0.000 }
gfCNCPoint4[24967] = {X 324.8079, Y 38.0635, Z -6.3333, A 0.000, B 0.000, C 0.000 }
gfCNCPoint4[24968] = {X 325.0860, Y 37.1389, Z -6.3333, A 0.000, B 0.000, C 0.000 }
gfCNCPoint4[24969] = {X 325.5408, Y 36.2871, Z -6.3333, A 0.000, B 0.000, C 0.000 }
gfCNCPoint4[24970] = {X 329.8000, Y 29.9189, Z -6.3333, A 0.000, B 0.000, C 0.000 }
gfCNCPoint4[24971] = {X 330.4881, Y 29.1146, Z -6.3333, A 0.000, B 0.000, C 0.000 }
gfCNCPoint4[24972] = {X 331.3333, Y 28.4776, Z -6.3333, A 0.000, B 0.000, C 0.000 }
gfCNCPoint4[24973] = {X 332.2961, Y 28.0378, Z -6.3333, A 0.000, B 0.000, C 0.000 }
gfCNCPoint4[24974] = {X 333.3310, Y 27.8160, Z -6.3333, A 0.000, B 0.000, C 0.000 }
gfCNCPoint4[24975] = {X 334.3894, Y 27.8225, Z -6.3333, A 0.000, B 0.000, C 0.000 }
gfCNCPoint4[24976] = {X 335.4215, Y 28.0570, Z -6.3333, A 0.000, B 0.000, C 0.000 }
gfCNCPoint4[24977] = {X 336.3787, Y 28.5085, Z -6.3333, A 0.000, B 0.000, C 0.000 }
gfCNCPoint4[24978] = {X 337.2161, Y 29.1559, Z -6.3333, A 0.000, B 0.000, C 0.000 }
gfCNCPoint4[24979] = {X 337.7864, Y 29.7052, Z -6.3333, A 0.000, B 0.000, C 0.000 }
gfCNCPoint4[24980] = {X 338.3558, Y 30.3610, Z -6.3333, A 0.000, B 0.000, C 0.000 }
gfCNCPoint4[24981] = {X 338.8000, Y 31.1075, Z -6.3333, A 0.000, B 0.000, C 0.000 }
gfCNCPoint4[24982] = {X 339.1047, Y 31.9208, Z -6.3333, A 0.000, B 0.000, C 0.000 }
gfCNCPoint4[24983] = {X 339.2605, Y 32.7753, Z -6.3333, A 0.000, B 0.000, C 0.000 }
gfCNCPoint4[24984] = {X 339.2623, Y 33.6438, Z -6.3333, A 0.000, B 0.000, C 0.000 }
gfCNCPoint4[24985] = {X 339.7987, Y 34.1193, Z -6.3333, A 0.000, B 0.000, C 0.000 }
gfCNCPoint4[24986] = {X 340.3478, Y 34.5800, Z -6.3333, A 0.000, B 0.000, C 0.000 }
gfCNCPoint4[24987] = {X 341.5551, Y 35.4252, Z -6.3333, A 0.000, B 0.000, C 0.000 }
gfCNCPoint4[24988] = {X 342.8733, Y 36.0843, Z -6.3333, A 0.000, B 0.000, C 0.000 }
gfCNCPoint4[24989] = {X 344.2739, Y 36.5428, Z -6.3333, A 0.000, B 0.000, C 0.000 }
gfCNCPoint4[24990] = {X 345.7267, Y 36.7909, Z -6.3333, A 0.000, B 0.000, C 0.000 }
gfCNCPoint4[24991] = {X 347.2001, Y 36.8232, Z -6.3333, A 0.000, B 0.000, C 0.000 }
gfCNCPoint4[24992] = {X 347.4897, Y 36.8082, Z -6.3333, A 0.000, B 0.000, C 0.000 }
gfCNCPoint4[24993] = {X 348.8392, Y 36.6270, Z -6.3333, A 0.000, B 0.000, C 0.000 }
gfCNCPoint4[24994] = {X 350.1412, Y 36.2284, Z -6.3333, A 0.000, B 0.000, C 0.000 }
gfCNCPoint4[24995] = {X 351.3609, Y 35.6232, Z -6.3333, A 0.000, B 0.000, C 0.000 }
gfCNCPoint4[24996] = {X 352.4658, Y 34.8275, Z -6.3333, A 0.000, B 0.000, C 0.000 }
gfCNCPoint4[24997] = {X 353.5667, Y 33.7579, Z -6.3333, A 0.000, B 0.000, C 0.000 }
gfCNCPoint4[24998] = {X 354.5195, Y 32.5544, Z -6.3333, A 0.000, B 0.000, C 0.000 }
gfCNCPoint4[24999] = {X 355.3080, Y 31.2374, Z -6.3333, A 0.000, B 0.000, C 0.000 }
gfCNCPoint4[25000] = {X 355.9189, Y 29.8293, Z -6.3333, A 0.000, B 0.000, C 0.000 }
gfCNCPoint4[25001] = {X 356.3419, Y 28.3538, Z -6.3333, A 0.000, B 0.000, C 0.000 }
gfCNCPoint4[25002] = {X 356.6064, Y 26.7186, Z -6.3333, A 0.000, B 0.000, C 0.000 }
gfCNCPoint4[25003] = {X 356.7141, Y 25.0657, Z -6.3333, A 0.000, B 0.000, C 0.000 }
gfCNCPoint4[25004] = {X 356.6640, Y 23.4100, Z -6.3333, A 0.000, B 0.000, C 0.000 }
gfCNCPoint4[25005] = {X 356.4566, Y 21.7666, Z -6.3333, A 0.000, B 0.000, C 0.000 }
gfCNCPoint4[25006] = {X 356.1199, Y 20.3210, Z -6.3333, A 0.000, B 0.000, C 0.000 }
gfCNCPoint4[25007] = {X 355.5962, Y 18.9321, Z -6.3333, A 0.000, B 0.000, C 0.000 }
gfCNCPoint4[25008] = {X 354.8947, Y 17.6240, Z -6.3333, A 0.000, B 0.000, C 0.000 }
gfCNCPoint4[25009] = {X 354.0274, Y 16.4193, Z -6.3333, A 0.000, B 0.000, C 0.000 }
gfCNCPoint4[25010] = {X 353.2099, Y 15.5484, Z -6.3333, A 0.000, B 0.000, C 0.000 }
gfCNCPoint4[25011] = {X 352.2795, Y 14.7994, Z -6.3333, A 0.000, B 0.000, C 0.000 }
gfCNCPoint4[25012] = {X 351.2542, Y 14.1866, Z -6.3333, A 0.000, B 0.000, C 0.000 }
gfCNCPoint4[25013] = {X 350.1538, Y 13.7220, Z -6.3333, A 0.000, B 0.000, C 0.000 }
gfCNCPoint4[25014] = {X 348.9995, Y 13.4146, Z -6.3333, A 0.000, B 0.000, C 0.000 }
gfCNCPoint4[25015] = {X 347.3622, Y 13.2068, Z -6.3333, A 0.000, B 0.000, C 0.000 }
gfCNCPoint4[25016] = {X 345.7117, Y 13.2115, Z -6.3333, A 0.000, B 0.000, C 0.000 }
gfCNCPoint4[25017] = {X 344.0755, Y 13.4284, Z -6.3333, A 0.000, B 0.000, C 0.000 }
gfCNCPoint4[25018] = {X 342.4808, Y 13.8541, Z -6.3333, A 0.000, B 0.000, C 0.000 }
gfCNCPoint4[25019] = {X 340.9542, Y 14.4814, Z -6.3333, A 0.000, B 0.000, C 0.000 }
gfCNCPoint4[25020] = {X 339.5209, Y 15.2999, Z -6.3333, A 0.000, B 0.000, C 0.000 }
gfCNCPoint4[25021] = {X 339.4271, Y 16.1855, Z -6.3333, A 0.000, B 0.000, C 0.000 }
gfCNCPoint4[25022] = {X 339.1739, Y 17.0394, Z -6.3333, A 0.000, B 0.000, C 0.000 }
gfCNCPoint4[25023] = {X 338.7698, Y 17.8330, Z -6.3333, A 0.000, B 0.000, C 0.000 }
gfCNCPoint4[25024] = {X 338.2281, Y 18.5399, Z -6.3333, A 0.000, B 0.000, C 0.000 }
gfCNCPoint4[25025] = {X 337.5670, Y 19.1366, Z -6.3333, A 0.000, B 0.000, C 0.000 }
gfCNCPoint4[25026] = {X 336.8400, Y 19.6716, Z -6.3333, A 0.000, B 0.000, C 0.000 }
gfCNCPoint4[25027] = {X 335.9171, Y 20.1909, Z -6.3333, A 0.000, B 0.000, C 0.000 }
gfCNCPoint4[25028] = {X 334.9039, Y 20.4988, Z -6.3333, A 0.000, B 0.000, C 0.000 }
gfCNCPoint4[25029] = {X 333.8481, Y 20.5809, Z -6.3333, A 0.000, B 0.000, C 0.000 }
gfCNCPoint4[25030] = {X 332.7995, Y 20.4334, Z -6.3333, A 0.000, B 0.000, C 0.000 }
gfCNCPoint4[25031] = {X 331.8074, Y 20.0631, Z -6.3333, A 0.000, B 0.000, C 0.000 }
gfCNCPoint4[25032] = {X 330.9186, Y 19.4875, Z -6.3333, A 0.000, B 0.000, C 0.000 }
gfCNCPoint4[25033] = {X 330.1748, Y 18.7338, Z -6.3333, A 0.000, B 0.000, C 0.000 }
gfCNCPoint4[25034] = {X 329.6111, Y 17.8373, Z -6.3333, A 0.000, B 0.000, C 0.000 }
gfCNCPoint4[25035] = {X 326.0906, Y 10.5950, Z -6.3333, A 0.000, B 0.000, C 0.000 }
gfCNCPoint4[25036] = {X 325.7555, Y 9.6856, Z -6.3333, A 0.000, B 0.000, C 0.000 }
gfCNCPoint4[25037] = {X 325.6067, Y 8.7279, Z -6.3333, A 0.000, B 0.000, C 0.000 }
gfCNCPoint4[25038] = {X 325.6502, Y 7.7596, Z -6.3333, A 0.000, B 0.000, C 0.000 }
gfCNCPoint4[25039] = {X 325.8842, Y 6.8191, Z -6.3333, A 0.000, B 0.000, C 0.000 }
gfCNCPoint4[25040] = {X 326.2994, Y 5.9434, Z -6.3333, A 0.000, B 0.000, C 0.000 }
gfCNCPoint4[25041] = {X 326.9295, Y 5.1131, Z -6.3333, A 0.000, B 0.000, C 0.000 }
gfCNCPoint4[25042] = {X 327.7216, Y 4.4356, Z -6.3333, A 0.000, B 0.000, C 0.000 }
gfCNCPoint4[25043] = {X 328.3968, Y 3.9733, Z -6.3333, A 0.000, B 0.000, C 0.000 }
gfCNCPoint4[25044] = {X 329.3292, Y 3.4829, Z -6.3333, A 0.000, B 0.000, C 0.000 }
gfCNCPoint4[25045] = {X 330.3452, Y 3.2041, Z -6.3333, A 0.000, B 0.000, C 0.000 }
gfCNCPoint4[25046] = {X 331.3973, Y 3.1498, Z -6.3333, A 0.000, B 0.000, C 0.000 }
gfCNCPoint4[25047] = {X 332.4365, Y 3.3226, Z -6.3333, A 0.000, B 0.000, C 0.000 }
gfCNCPoint4[25048] = {X 333.3723, Y 2.7963, Z -6.3333, A 0.000, B 0.000, C 0.000 }
gfCNCPoint4[25049] = {X 334.3269, Y 2.3049, Z -6.3333, A 0.000, B 0.000, C 0.000 }
gfCNCPoint4[25050] = {X 334.5387, Y 2.7357, Z -6.3333, A 0.000, B 0.000, C 0.000 }
gfCNCPoint4[25051] = {X 335.1908, Y 2.4252, Z -6.3333, A 0.000, B 0.000, C 0.000 }
gfCNCPoint4[25052] = {X 335.8505, Y 2.1314, Z -6.3333, A 0.000, B 0.000, C 0.000 }
gfCNCPoint4[25053] = {X 336.0151, Y 2.0603, Z -6.3333, A 0.000, B 0.000, C 0.000 }
gfCNCPoint4[25054] = {X 338.1014, Y 1.2621, Z -6.3333, A 0.000, B 0.000, C 0.000 }
gfCNCPoint4[25055] = {X 340.2478, Y 0.6433, Z -6.3333, A 0.000, B 0.000, C 0.000 }
gfCNCPoint4[25056] = {X 342.4388, Y 0.2084, Z -6.3333, A 0.000, B 0.000, C 0.000 }
gfCNCPoint4[25057] = {X 344.6588, Y -0.0396, Z -6.3333, A 0.000, B 0.000, C 0.000 }
gfCNCPoint4[25058] = {X 346.8919, Y -0.0989, Z -6.3333, A 0.000, B 0.000, C 0.000 }
gfCNCPoint4[25059] = {X 349.1219, Y 0.0310, Z -6.3333, A 0.000, B 0.000, C 0.000 }
gfCNCPoint4[25060] = {X 351.3329, Y 0.3491, Z -6.3333, A 0.000, B 0.000, C 0.000 }
gfCNCPoint4[25061] = {X 351.8887, Y 0.4533, Z -6.3333, A 0.000, B 0.000, C 0.000 }
gfCNCPoint4[25062] = {X 353.8464, Y 0.9458, Z -6.3333, A 0.000, B 0.000, C 0.000 }
gfCNCPoint4[25063] = {X 355.7482, Y 1.6232, Z -6.3333, A 0.000, B 0.000, C 0.000 }
gfCNCPoint4[25064] = {X 357.5764, Y 2.4793, Z -6.3333, A 0.000, B 0.000, C 0.000 }
gfCNCPoint4[25065] = {X 359.3145, Y 3.5063, Z -6.3333, A 0.000, B 0.000, C 0.000 }
gfCNCPoint4[25066] = {X 360.9464, Y 4.6947, Z -6.3333, A 0.000, B 0.000, C 0.000 }
gfCNCPoint4[25067] = {X 362.4573, Y 6.0337, Z -6.3333, A 0.000, B 0.000, C 0.000 }
gfCNCPoint4[25068] = {X 363.8332, Y 7.5110, Z -6.3333, A 0.000, B 0.000, C 0.000 }
gfCNCPoint4[25069] = {X 365.1885, Y 9.2728, Z -6.3333, A 0.000, B 0.000, C 0.000 }
gfCNCPoint4[25070] = {X 366.3832, Y 11.1473, Z -6.3333, A 0.000, B 0.000, C 0.000 }
gfCNCPoint4[25071] = {X 367.4079, Y 13.1199, Z -6.3333, A 0.000, B 0.000, C 0.000 }
gfCNCPoint4[25072] = {X 368.2546, Y 15.1751, Z -6.3333, A 0.000, B 0.000, C 0.000 }
gfCNCPoint4[25073] = {X 368.9169, Y 17.2970, Z -6.3333, A 0.000, B 0.000, C 0.000 }
gfCNCPoint4[25074] = {X 369.3894, Y 19.4690, Z -6.3333, A 0.000, B 0.000, C 0.000 }
gfCNCPoint4[25075] = {X 369.7212, Y 21.8433, Z -6.3333, A 0.000, B 0.000, C 0.000 }
gfCNCPoint4[25076] = {X 369.8733, Y 24.2358, Z -6.3333, A 0.000, B 0.000, C 0.000 }
gfCNCPoint4[25077] = {X 369.8449, Y 26.6330, Z -6.3333, A 0.000, B 0.000, C 0.000 }
gfCNCPoint4[25078] = {X 369.6361, Y 29.0212, Z -6.3333, A 0.000, B 0.000, C 0.000 }
gfCNCPoint4[25079] = {X 369.2481, Y 31.3870, Z -6.3333, A 0.000, B 0.000, C 0.000 }
gfCNCPoint4[25080] = {X 368.7224, Y 33.4980, Z -6.3333, A 0.000, B 0.000, C 0.000 }
gfCNCPoint4[25081] = {X 368.0123, Y 35.5544, Z -6.3333, A 0.000, B 0.000, C 0.000 }
gfCNCPoint4[25082] = {X 367.1234, Y 37.5400, Z -6.3333, A 0.000, B 0.000, C 0.000 }
gfCNCPoint4[25083] = {X 366.0626, Y 39.4394, Z -6.3333, A 0.000, B 0.000, C 0.000 }
gfCNCPoint4[25084] = {X 364.8382, Y 41.2377, Z -6.3333, A 0.000, B 0.000, C 0.000 }
gfCNCPoint4[25085] = {X 364.7204, Y 41.3988, Z -6.3333, A 0.000, B 0.000, C 0.000 }
gfCNCPoint4[25086] = {X 363.4201, Y 42.9675, Z -6.3333, A 0.000, B 0.000, C 0.000 }
gfCNCPoint4[25087] = {X 361.9805, Y 44.4097, Z -6.3333, A 0.000, B 0.000, C 0.000 }
gfCNCPoint4[25088] = {X 360.4141, Y 45.7129, Z -6.3333, A 0.000, B 0.000, C 0.000 }
gfCNCPoint4[25089] = {X 358.7341, Y 46.8660, Z -6.3333, A 0.000, B 0.000, C 0.000 }
gfCNCPoint4[25090] = {X 356.9549, Y 47.8592, Z -6.3333, A 0.000, B 0.000, C 0.000 }
gfCNCPoint4[25091] = {X 356.2499, Y 48.1928, Z -6.3333, A 0.000, B 0.000, C 0.000 }
gfCNCPoint4[25092] = {X 354.0456, Y 49.0152, Z -6.3333, A 0.000, B 0.000, C 0.000 }
gfCNCPoint4[25093] = {X 351.7691, Y 49.6091, Z -6.3333, A 0.000, B 0.000, C 0.000 }
gfCNCPoint4[25094] = {X 349.4439, Y 49.9685, Z -6.3333, A 0.000, B 0.000, C 0.000 }
gfCNCPoint4[25095] = {X 347.0943, Y 50.0896, Z -6.3333, A 0.000, B 0.000, C 0.000 }
gfCNCPoint4[25096] = {X 345.0202, Y 50.0544, Z -6.3333, A 0.000, B 0.000, C 0.000 }
gfCNCPoint4[25097] = {X 342.9569, Y 49.8395, Z -6.3333, A 0.000, B 0.000, C 0.000 }
gfCNCPoint4[25098] = {X 340.9200, Y 49.4464, Z -6.3333, A 0.000, B 0.000, C 0.000 }
gfCNCPoint4[25099] = {X 338.9249, Y 48.8780, Z -6.3333, A 0.000, B 0.000, C 0.000 }
gfCNCPoint4[25100] = {X 336.9867, Y 48.1387, Z -6.3333, A 0.000, B 0.000, C 0.000 }
gfCNCPoint4[25101] = {X 335.1198, Y 47.2341, Z -6.3333, A 0.000, B 0.000, C 0.000 }
gfCNCPoint4[25102] = {X 333.5418, Y 46.2597, Z -6.3333, A 0.000, B 0.000, C 0.000 }
gfCNCPoint4[25103] = {X 332.0438, Y 45.1662, Z -6.3333, A 0.000, B 0.000, C 0.000 }
gfCNCPoint4[25104] = {X 330.6347, Y 43.9603, Z -6.3333, A 0.000, B 0.000, C 0.000 }
gfCNCPoint4[25105] = {X 329.6761, Y 43.9518, Z -6.3333, A 0.000, B 0.000, C 0.000 }
gfCNCPoint4[25106] = {X 328.7421, Y 43.7359, Z -6.3333, A 0.000, B 0.000, C 0.000 }
gfCNCPoint4[25107] = {X 327.8770, Y 43.3228, Z -6.3333, A 0.000, B 0.000, C 0.000 }
gfCNCPoint4[25108] = {X 327.1220, Y 42.7322, Z -6.3333, A 0.000, B 0.000, C 0.000 }
gfCNCPoint4[25109] = {X 326.5249, Y 42.1498, Z -6.3333, A 0.000, B 0.000, C 0.000 }
gfCNCPoint4[25110] = {X 325.8848, Y 41.3619, Z -6.3333, A 0.000, B 0.000, C 0.000 }
gfCNCPoint4[25111] = {X 325.4424, Y 40.4483, Z -6.3333, A 0.000, B 0.000, C 0.000 }
gfCNCPoint4[25112] = {X 325.2210, Y 39.4576, Z -6.3333, A 0.000, B 0.000, C 0.000 }
gfCNCPoint4[25113] = {X 325.2326, Y 38.4426, Z -6.3333, A 0.000, B 0.000, C 0.000 }
gfCNCPoint4[25114] = {X 325.4765, Y 37.4572, Z -6.3333, A 0.000, B 0.000, C 0.000 }
gfCNCPoint4[25115] = {X 325.9398, Y 36.5539, Z -6.3333, A 0.000, B 0.000, C 0.000 }
gfCNCPoint4[25116] = {X 330.1988, Y 30.1861, Z -6.3333, A 0.000, B 0.000, C 0.000 }
gfCNCPoint4[25117] = {X 330.8195, Y 29.4619, Z -6.3333, A 0.000, B 0.000, C 0.000 }
gfCNCPoint4[25118] = {X 331.5816, Y 28.8884, Z -6.3333, A 0.000, B 0.000, C 0.000 }
gfCNCPoint4[25119] = {X 332.4495, Y 28.4927, Z -6.3333, A 0.000, B 0.000, C 0.000 }
gfCNCPoint4[25120] = {X 333.3822, Y 28.2932, Z -6.3333, A 0.000, B 0.000, C 0.000 }
gfCNCPoint4[25121] = {X 334.3359, Y 28.2995, Z -6.3333, A 0.000, B 0.000, C 0.000 }
gfCNCPoint4[25122] = {X 335.2660, Y 28.5111, Z -6.3333, A 0.000, B 0.000, C 0.000 }
gfCNCPoint4[25123] = {X 336.1285, Y 28.9182, Z -6.3333, A 0.000, B 0.000, C 0.000 }
gfCNCPoint4[25124] = {X 336.8831, Y 29.5016, Z -6.3333, A 0.000, B 0.000, C 0.000 }
gfCNCPoint4[25125] = {X 337.4845, Y 30.0811, Z -6.3333, A 0.000, B 0.000, C 0.000 }
gfCNCPoint4[25126] = {X 338.1269, Y 30.8797, Z -6.3333, A 0.000, B 0.000, C 0.000 }
gfCNCPoint4[25127] = {X 338.5672, Y 31.8052, Z -6.3333, A 0.000, B 0.000, C 0.000 }
gfCNCPoint4[25128] = {X 338.7814, Y 32.8075, Z -6.3333, A 0.000, B 0.000, C 0.000 }
gfCNCPoint4[25129] = {X 338.7580, Y 33.8321, Z -6.3333, A 0.000, B 0.000, C 0.000 }
gfCNCPoint4[25130] = {X 339.3922, Y 34.4022, Z -6.3333, A 0.000, B 0.000, C 0.000 }
gfCNCPoint4[25131] = {X 340.0443, Y 34.9519, Z -6.3333, A 0.000, B 0.000, C 0.000 }
gfCNCPoint4[25132] = {X 341.3094, Y 35.8376, Z -6.3333, A 0.000, B 0.000, C 0.000 }
gfCNCPoint4[25133] = {X 342.6908, Y 36.5282, Z -6.3333, A 0.000, B 0.000, C 0.000 }
gfCNCPoint4[25134] = {X 344.1585, Y 37.0087, Z -6.3333, A 0.000, B 0.000, C 0.000 }
gfCNCPoint4[25135] = {X 345.6809, Y 37.2687, Z -6.3333, A 0.000, B 0.000, C 0.000 }
gfCNCPoint4[25136] = {X 347.2249, Y 37.3025, Z -6.3333, A 0.000, B 0.000, C 0.000 }
gfCNCPoint4[25137] = {X 347.5145, Y 37.2875, Z -6.3333, A 0.000, B 0.000, C 0.000 }
gfCNCPoint4[25138] = {X 348.9417, Y 37.0959, Z -6.3333, A 0.000, B 0.000, C 0.000 }
gfCNCPoint4[25139] = {X 350.3187, Y 36.6744, Z -6.3333, A 0.000, B 0.000, C 0.000 }
gfCNCPoint4[25140] = {X 351.6087, Y 36.0343, Z -6.3333, A 0.000, B 0.000, C 0.000 }
gfCNCPoint4[25141] = {X 352.7772, Y 35.1928, Z -6.3333, A 0.000, B 0.000, C 0.000 }
gfCNCPoint4[25142] = {X 353.9231, Y 34.0794, Z -6.3333, A 0.000, B 0.000, C 0.000 }
gfCNCPoint4[25143] = {X 354.9147, Y 32.8267, Z -6.3333, A 0.000, B 0.000, C 0.000 }
gfCNCPoint4[25144] = {X 355.7354, Y 31.4559, Z -6.3333, A 0.000, B 0.000, C 0.000 }
gfCNCPoint4[25145] = {X 356.3711, Y 29.9902, Z -6.3333, A 0.000, B 0.000, C 0.000 }
gfCNCPoint4[25146] = {X 356.8112, Y 28.4543, Z -6.3333, A 0.000, B 0.000, C 0.000 }
gfCNCPoint4[25147] = {X 357.0833, Y 26.7727, Z -6.3333, A 0.000, B 0.000, C 0.000 }
gfCNCPoint4[25148] = {X 357.1940, Y 25.0729, Z -6.3333, A 0.000, B 0.000, C 0.000 }
gfCNCPoint4[25149] = {X 357.1423, Y 23.3702, Z -6.3333, A 0.000, B 0.000, C 0.000 }
gfCNCPoint4[25150] = {X 356.9288, Y 21.6802, Z -6.3333, A 0.000, B 0.000, C 0.000 }
gfCNCPoint4[25151] = {X 356.5771, Y 20.1748, Z -6.3333, A 0.000, B 0.000, C 0.000 }
gfCNCPoint4[25152] = {X 356.0310, Y 18.7287, Z -6.3333, A 0.000, B 0.000, C 0.000 }
gfCNCPoint4[25153] = {X 355.2999, Y 17.3666, Z -6.3333, A 0.000, B 0.000, C 0.000 }
gfCNCPoint4[25154] = {X 354.3964, Y 16.1123, Z -6.3333, A 0.000, B 0.000, C 0.000 }
gfCNCPoint4[25155] = {X 353.5334, Y 15.1938, Z -6.3333, A 0.000, B 0.000, C 0.000 }
gfCNCPoint4[25156] = {X 352.5515, Y 14.4038, Z -6.3333, A 0.000, B 0.000, C 0.000 }
gfCNCPoint4[25157] = {X 351.4695, Y 13.7576, Z -6.3333, A 0.000, B 0.000, C 0.000 }
gfCNCPoint4[25158] = {X 350.3084, Y 13.2676, Z -6.3333, A 0.000, B 0.000, C 0.000 }
gfCNCPoint4[25159] = {X 349.0905, Y 12.9433, Z -6.3333, A 0.000, B 0.000, C 0.000 }
gfCNCPoint4[25160] = {X 347.3478, Y 12.7251, Z -6.3333, A 0.000, B 0.000, C 0.000 }
gfCNCPoint4[25161] = {X 345.5916, Y 12.7388, Z -6.3333, A 0.000, B 0.000, C 0.000 }
gfCNCPoint4[25162] = {X 343.8525, Y 12.9841, Z -6.3333, A 0.000, B 0.000, C 0.000 }
gfCNCPoint4[25163] = {X 342.1610, Y 13.4567, Z -6.3333, A 0.000, B 0.000, C 0.000 }
gfCNCPoint4[25164] = {X 340.5466, Y 14.1483, Z -6.3333, A 0.000, B 0.000, C 0.000 }
gfCNCPoint4[25165] = {X 339.0376, Y 15.0469, Z -6.3333, A 0.000, B 0.000, C 0.000 }
gfCNCPoint4[25166] = {X 338.9895, Y 15.9047, Z -6.3333, A 0.000, B 0.000, C 0.000 }
gfCNCPoint4[25167] = {X 338.7757, Y 16.7368, Z -6.3333, A 0.000, B 0.000, C 0.000 }
gfCNCPoint4[25168] = {X 338.4042, Y 17.5115, Z -6.3333, A 0.000, B 0.000, C 0.000 }
gfCNCPoint4[25169] = {X 337.8892, Y 18.1993, Z -6.3333, A 0.000, B 0.000, C 0.000 }
gfCNCPoint4[25170] = {X 337.2504, Y 18.7738, Z -6.3333, A 0.000, B 0.000, C 0.000 }
gfCNCPoint4[25171] = {X 336.5606, Y 19.2813, Z -6.3333, A 0.000, B 0.000, C 0.000 }
gfCNCPoint4[25172] = {X 335.7284, Y 19.7495, Z -6.3333, A 0.000, B 0.000, C 0.000 }
gfCNCPoint4[25173] = {X 334.8148, Y 20.0271, Z -6.3333, A 0.000, B 0.000, C 0.000 }
gfCNCPoint4[25174] = {X 333.8628, Y 20.1012, Z -6.3333, A 0.000, B 0.000, C 0.000 }
gfCNCPoint4[25175] = {X 332.9173, Y 19.9681, Z -6.3333, A 0.000, B 0.000, C 0.000 }
gfCNCPoint4[25176] = {X 332.0228, Y 19.6341, Z -6.3333, A 0.000, B 0.000, C 0.000 }
gfCNCPoint4[25177] = {X 331.2213, Y 19.1151, Z -6.3333, A 0.000, B 0.000, C 0.000 }
gfCNCPoint4[25178] = {X 330.5507, Y 18.4353, Z -6.3333, A 0.000, B 0.000, C 0.000 }
gfCNCPoint4[25179] = {X 330.0425, Y 17.6269, Z -6.3333, A 0.000, B 0.000, C 0.000 }
gfCNCPoint4[25180] = {X 326.5223, Y 10.3852, Z -6.3333, A 0.000, B 0.000, C 0.000 }
gfCNCPoint4[25181] = {X 326.2154, Y 9.5469, Z -6.3333, A 0.000, B 0.000, C 0.000 }
gfCNCPoint4[25182] = {X 326.0841, Y 8.6639, Z -6.3333, A 0.000, B 0.000, C 0.000 }
gfCNCPoint4[25183] = {X 326.1338, Y 7.7725, Z -6.3333, A 0.000, B 0.000, C 0.000 }
gfCNCPoint4[25184] = {X 326.3623, Y 6.9096, Z -6.3333, A 0.000, B 0.000, C 0.000 }
gfCNCPoint4[25185] = {X 326.7603, Y 6.1105, Z -6.3333, A 0.000, B 0.000, C 0.000 }
gfCNCPoint4[25186] = {X 327.3114, Y 5.4082, Z -6.3333, A 0.000, B 0.000, C 0.000 }
gfCNCPoint4[25187] = {X 327.9929, Y 4.8316, Z -6.3333, A 0.000, B 0.000, C 0.000 }
gfCNCPoint4[25188] = {X 328.6647, Y 4.3715, Z -6.3333, A 0.000, B 0.000, C 0.000 }
gfCNCPoint4[25189] = {X 329.5522, Y 3.9112, Z -6.3333, A 0.000, B 0.000, C 0.000 }
gfCNCPoint4[25190] = {X 330.5207, Y 3.6631, Z -6.3333, A 0.000, B 0.000, C 0.000 }
gfCNCPoint4[25191] = {X 331.5202, Y 3.6401, Z -6.3333, A 0.000, B 0.000, C 0.000 }
gfCNCPoint4[25192] = {X 332.4991, Y 3.8433, Z -6.3333, A 0.000, B 0.000, C 0.000 }
gfCNCPoint4[25193] = {X 333.5077, Y 3.2688, Z -6.3333, A 0.000, B 0.000, C 0.000 }
gfCNCPoint4[25194] = {X 334.5387, Y 2.7357, Z -6.3333, A 0.000, B 0.000, C 0.000 }
gfCNCPoint4[25195] = {X 334.3269, Y 2.3049, Z -6.3333, A 0.000, B 0.000, C 0.000 }
